KUKA KRL program: MyProgram_231().src

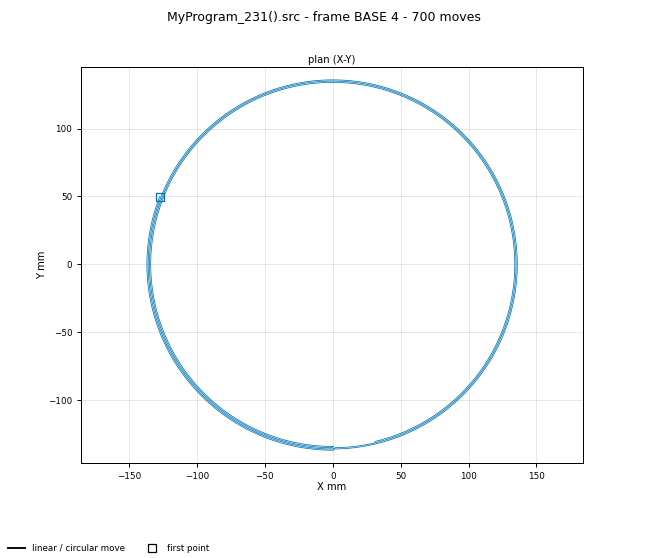
[picture p0: tool path of MyProgram_231().src in frame BASE 4, 700 of 700 moves have a stored position in this frame; points joined in program order, loops and branches not executed]
&ACCESS RVP
&REL 1
&PARAM TEMPLATE = C:\KRC\Roboter\Template\vorgabe
&PARAM EDITMASK = *
DEF MyProgram_231()
; ---- Setting reference (Base) ----
$BASE = BASE_DATA[4]

; --------------------------
; ---- Setting tool (TCP) ----
$TOOL = TOOL_DATA[3]
; --------------------------

$VEL.CP = VEL_APROX_PRINT
Startdeposition()
$VEL.CP = VEL_PRINT
LIN {X -127.3745,Y 49.9123,Z 158,A 155.4211,B 24.9582,C -1.4929,E1 24.8505,E2 291.1488} C_DIS
LIN {X -128.4799,Y 46.9966,Z 158,A 156.8322,B 24.9582,C -1.4941,E1 24.8491,E2 289.7271} C_DIS
LIN {X -130.1138,Y 42.2637,Z 158,A 158.8681,B 24.9587,C -1.4842,E1 24.8473,E2 287.7029} C_DIS
LIN {X -131.1004,Y 39.0966,Z 158,A 160.3394,B 24.9587,C -1.4839,E1 24.8461,E2 286.224} C_DIS
LIN {X -132.2192,Y 35.1211,Z 158,A 161.9803,B 24.9593,C -1.4738,E1 24.8449,E2 284.5976} C_DIS
LIN {X -133.0966,Y 31.6367,Z 158,A 163.554,B 24.9593,C -1.4724,E1 24.8439,E2 283.0182} C_DIS
LIN {X -133.994,Y 27.5885,Z 158,A 165.3357,B 24.9596,C -1.4689,E1 24.8428,E2 281.2342} C_DIS
LIN {X -134.7246,Y 23.7659,Z 158,A 166.9993,B 24.9598,C -1.4652,E1 24.842,E2 279.5695} C_DIS
LIN {X -135.3385,Y 19.9835,Z 158,A 168.5128,B 24.9603,C -1.4553,E1 24.8414,E2 278.0706} C_DIS
LIN {X -135.7642,Y 16.8509,Z 158,A 169.8487,B 24.9605,C -1.4515,E1 24.8409,E2 276.7357} C_DIS
LIN {X -136.156,Y 13.3069,Z 158,A 171.4307,B 24.9605,C -1.4511,E1 24.8404,E2 275.1454} C_DIS
LIN {X -136.4953,Y 9.2216,Z 158,A 173.2066,B 24.9607,C -1.4483,E1 24.8401,E2 273.3653} C_DIS
LIN {X -136.7019,Y 5.2983,Z 158,A 174.7382,B 24.9613,C -1.4371,E1 24.8399,E2 271.8512} C_DIS
LIN {X -136.7995,Y 1.3383,Z 158,A 176.4739,B 24.9613,C -1.4355,E1 24.8398,E2 270.1089} C_DIS
LIN {X -136.7858,Y -2.2665,Z 158,A 177.9865,B 24.9617,C -1.4306,E1 24.8398,E2 268.5987} C_DIS
LIN {X -136.6643,Y -6.2262,Z 158,A 179.6239,B 24.962,C -1.424,E1 24.84,E2 266.9672} C_DIS
LIN {X -136.4748,Y -9.5029,Z 158,A -178.911,B 24.962,C -1.4241,E1 24.8403,E2 265.4932} C_DIS
LIN {X -136.1015,Y -13.8716,Z 158,A -177.0261,B 24.9622,C -1.4205,E1 24.8408,E2 263.6055} C_DIS
LIN {X -135.632,Y -17.8725,Z 158,A -175.4762,B 24.9629,C -1.4081,E1 24.8413,E2 262.076} C_DIS
LIN {X -135.0766,Y -21.687,Z 158,A -173.7107,B 24.9627,C -1.4105,E1 24.8421,E2 260.2943} C_DIS
LIN {X -134.5265,Y -24.8732,Z 158,A -172.3224,B 24.9629,C -1.4078,E1 24.8428,E2 258.904} C_DIS
LIN {X -133.6444,Y -29.2358,Z 158,A -170.5745,B 24.9635,C -1.396,E1 24.8438,E2 257.174} C_DIS
LIN {X -132.6945,Y -33.2823,Z 158,A -168.7848,B 24.9637,C -1.393,E1 24.8449,E2 255.3811} C_DIS
LIN {X -130.9297,Y -39.6606,Z 158,A -166.0195,B 24.9641,C -1.3839,E1 24.8471,E2 252.6213} C_DIS
LIN {X -129.8846,Y -42.9585,Z 158,A -164.5726,B 24.9644,C -1.3794,E1 24.8483,E2 251.1769} C_DIS
LIN {X -128.7046,Y -46.3735,Z 158,A -163.0102,B 24.9644,C -1.3773,E1 24.8498,E2 249.6107} C_DIS
LIN {X -127.0686,Y -50.6869,Z 158,A -161.1504,B 24.965,C -1.3677,E1 24.8516,E2 247.7632} C_DIS
LIN {X -125.8439,Y -53.6576,Z 158,A -159.7893,B 24.9651,C -1.3645,E1 24.8531,E2 246.4022} C_DIS
LIN {X -121.9807,Y -61.9359,Z 158,A -155.9432,B 24.9656,C -1.3543,E1 24.8577,E2 242.5594} C_DIS
LIN {X -119.7997,Y -66.0603,Z 158,A -153.8465,B 24.9656,C -1.3561,E1 24.8605,E2 240.4475} C_DIS
LIN {X -117.4088,Y -70.2217,Z 158,A -151.8184,B 24.9658,C -1.3515,E1 24.8634,E2 238.4198} C_DIS
LIN {X -114.9649,Y -74.1559,Z 158,A -149.8617,B 24.966,C -1.3472,E1 24.8663,E2 236.4634} C_DIS
LIN {X -112.5613,Y -77.756,Z 158,A -148.04,B 24.9662,C -1.3429,E1 24.8691,E2 234.643} C_DIS
LIN {X -109.8954,Y -81.4797,Z 158,A -146.1227,B 24.9665,C -1.338,E1 24.8723,E2 232.7281} C_DIS
LIN {X -107.338,Y -84.8209,Z 158,A -144.3319,B 24.9666,C -1.3351,E1 24.8754,E2 230.9357} C_DIS
LIN {X -104.393,Y -88.4196,Z 158,A -142.0462,B 24.966,C -1.348,E1 24.8795,E2 228.6087} C_DIS
LIN {X -101.6067,Y -91.6087,Z 158,A -140.6091,B 24.9671,C -1.3263,E1 24.8821,E2 227.2167} C_DIS
LIN {X -98.4941,Y -94.9467,Z 158,A -138.4408,B 24.9666,C -1.3354,E1 24.8864,E2 225.0174} C_DIS
LIN {X -95.9147,Y -97.5514,Z 158,A -137.1932,B 24.9675,C -1.3171,E1 24.8888,E2 223.8082} C_DIS
LIN {X -92.7603,Y -100.5557,Z 158,A -135.4258,B 24.9678,C -1.3103,E1 24.8924,E2 222.0497} C_DIS
LIN {X -85.315,Y -106.945,Z 158,A -131.294,B 24.9682,C -1.3032,E1 24.9012,E2 217.9188} C_DIS
LIN {X -82.1496,Y -109.3957,Z 158,A -129.5135,B 24.9681,C -1.3056,E1 24.9051,E2 216.1262} C_DIS
LIN {X -78.4965,Y -112.0463,Z 158,A -127.6003,B 24.9681,C -1.3035,E1 24.9095,E2 214.2114} C_DIS
LIN {X -74.8596,Y -114.5081,Z 158,A -125.7445,B 24.9683,C -1.3014,E1 24.9138,E2 212.3545} C_DIS
LIN {X -71.0332,Y -116.9198,Z 158,A -123.9031,B 24.9686,C -1.2956,E1 24.9182,E2 210.521} C_DIS
LIN {X -67.4593,Y -119.0179,Z 158,A -122.1621,B 24.9686,C -1.2934,E1 24.9224,E2 208.7802} C_DIS
LIN {X -63.8309,Y -121,Z 158,A -120.5227,B 24.969,C -1.2862,E1 24.9264,E2 207.1533} C_DIS
LIN {X -60.8744,Y -122.5145,Z 158,A -119.0759,B 24.969,C -1.2873,E1 24.93,E2 205.6999} C_DIS
LIN {X -51.1886,Y -126.8664,Z 158,A -114.6733,B 24.9693,C -1.2798,E1 24.9413,E2 201.3046} C_DIS
LIN {X -47.6136,Y -128.2516,Z 158,A -112.9917,B 24.9693,C -1.2823,E1 24.9457,E2 199.6137} C_DIS
LIN {X -43.4067,Y -129.7354,Z 158,A -111.2356,B 24.9696,C -1.2746,E1 24.9503,E2 197.8723} C_DIS
LIN {X -40.213,Y -130.7606,Z 158,A -109.8746,B 24.9697,C -1.2712,E1 24.9539,E2 196.517} C_DIS
LIN {X -37.5338,Y -131.5565,Z 158,A -108.4891,B 24.9692,C -1.2819,E1 24.9577,E2 195.1038} C_DIS
LIN {X -33.8507,Y -132.5503,Z 158,A -106.9831,B 24.9695,C -1.276,E1 24.9617,E2 193.6096} C_DIS
LIN {X -30.4717,Y -133.3675,Z 158,A -105.5552,B 24.9696,C -1.2737,E1 24.9656,E2 192.1852} C_DIS
LIN {X -27.3724,Y -134.038,Z 158,A -104.1952,B 24.9696,C -1.2748,E1 24.9693,E2 190.821} C_DIS
LIN {X -23.966,Y -134.6888,Z 158,A -102.7439,B 24.9696,C -1.2742,E1 24.9733,E2 189.3695} C_DIS
LIN {X -19.992,Y -135.3373,Z 158,A -100.9635,B 24.9694,C -1.2788,E1 24.9782,E2 187.5768} C_DIS
LIN {X -11.9765,Y -136.28,Z 158,A -97.5382,B 24.9693,C -1.2808,E1 24.9878,E2 184.1446} C_DIS
LIN {X -7.2873,Y -136.611,Z 158,A -95.6653,B 24.9695,C -1.2756,E1 24.9929,E2 182.2833} C_DIS
LIN {X 0.1481,Y -136.8059,Z 158,A -92.6859,B 24.9699,C -1.2686,E1 25.0012,E2 179.3202} C_DIS
LIN {X 0.1481,Y -136.8059,Z 158,A -92.6859,B 24.9699,C -1.2686,E1 25.0012,E2 179.3202} C_DIS
Enddeposition()
LIN {X 0.9433,Y -135.864,Z 158,A -91.8366,B 24.2391,C -1.1592,E1 24.2683,E2 178.6405} C_DIS
Startdeposition()
$VEL.CP = VEL_PRINT
LIN {X -4.3433,Y -135.807,Z 158,A -94.8507,B 24.241,C -1.1174,E1 24.2596,E2 181.7565} C_DIS
LIN {X -7.4971,Y -135.6699,Z 158,A -96.5948,B 24.2419,C -1.096,E1 24.2546,E2 183.5533} C_DIS
LIN {X -11.0273,Y -135.4276,Z 158,A -97.7763,B 24.2412,C -1.112,E1 24.2514,E2 184.6963} C_DIS
LIN {X -15.1641,Y -135.0278,Z 158,A -99.4494,B 24.241,C -1.1163,E1 24.2467,E2 186.3599} C_DIS
LIN {X -18.8588,Y -134.5605,Z 158,A -101.1029,B 24.2412,C -1.1124,E1 24.2421,E2 188.0243} C_DIS
LIN {X -22.4613,Y -134.0057,Z 158,A -102.5865,B 24.2411,C -1.1156,E1 24.2381,E2 189.5014} C_DIS
LIN {X -25.8541,Y -133.393,Z 158,A -104.0291,B 24.2411,C -1.1167,E1 24.2341,E2 190.9429} C_DIS
LIN {X -29.7466,Y -132.5799,Z 158,A -105.7981,B 24.2411,C -1.1128,E1 24.2292,E2 192.7237} C_DIS
LIN {X -33.6182,Y -131.6505,Z 158,A -107.339,B 24.2408,C -1.1208,E1 24.2251,E2 194.2473} C_DIS
LIN {X -36.7276,Y -130.817,Z 158,A -108.7487,B 24.2409,C -1.119,E1 24.2213,E2 195.6636} C_DIS
LIN {X -39.7605,Y -129.9272,Z 158,A -110.1344,B 24.2409,C -1.1173,E1 24.2176,E2 197.0559} C_DIS
LIN {X -43.4862,Y -128.7294,Z 158,A -111.7492,B 24.2409,C -1.1204,E1 24.2133,E2 198.6661} C_DIS
LIN {X -47.3237,Y -127.3678,Z 158,A -113.58,B 24.241,C -1.1162,E1 24.2085,E2 200.511} C_DIS
LIN {X -51.0417,Y -125.9237,Z 158,A -115.147,B 24.2407,C -1.1237,E1 24.2044,E2 202.0632} C_DIS
LIN {X -56.4466,Y -123.5966,Z 158,A -117.6806,B 24.2407,C -1.1238,E1 24.1979,E2 204.6028} C_DIS
LIN {X -58.9215,Y -122.435,Z 158,A -118.8087,B 24.2406,C -1.1265,E1 24.1951,E2 205.7274} C_DIS
LIN {X -62.0587,Y -120.8754,Z 158,A -120.4233,B 24.2408,C -1.1215,E1 24.191,E2 207.3586} C_DIS
LIN {X -66.2441,Y -118.6353,Z 158,A -122.1842,B 24.2402,C -1.1363,E1 24.1868,E2 209.0885} C_DIS
LIN {X -69.0311,Y -117.0352,Z 158,A -124.0916,B 24.2413,C -1.1108,E1 24.182,E2 211.0643} C_DIS
LIN {X -72.4789,Y -114.9316,Z 158,A -125.2628,B 24.24,C -1.1399,E1 24.1794,E2 212.1682} C_DIS
LIN {X -75.4383,Y -113.0112,Z 158,A -126.9217,B 24.2403,C -1.1337,E1 24.1755,E2 213.8477} C_DIS
LIN {X -79.0416,Y -110.521,Z 158,A -128.8017,B 24.2403,C -1.1352,E1 24.1712,E2 215.7307} C_DIS
LIN {X -82.7672,Y -107.7596,Z 158,A -130.7512,B 24.24,C -1.1391,E1 24.1668,E2 217.6781} C_DIS
LIN {X -86.0862,Y -105.1268,Z 158,A -132.9637,B 24.2408,C -1.1215,E1 24.1619,E2 219.9422} C_DIS
LIN {X -89.3998,Y -102.3233,Z 158,A -134.2995,B 24.2396,C -1.1494,E1 24.1593,E2 221.215} C_DIS
LIN {X -91.7357,Y -100.2353,Z 158,A -135.6918,B 24.2396,C -1.1486,E1 24.1564,E2 222.6151} C_DIS
LIN {X -94.8002,Y -97.3424,Z 158,A -137.6191,B 24.2398,C -1.145,E1 24.1524,E2 224.5595} C_DIS
LIN {X -97.5363,Y -94.5999,Z 158,A -139.1597,B 24.2394,C -1.1531,E1 24.1495,E2 226.087} C_DIS
LIN {X -100.5896,Y -91.3466,Z 158,A -140.8497,B 24.2388,C -1.1668,E1 24.1463,E2 227.7514} C_DIS
LIN {X -103.1897,Y -88.3994,Z 158,A -142.447,B 24.2385,C -1.1736,E1 24.1434,E2 229.3394} C_DIS
LIN {X -105.0465,Y -86.1845,Z 158,A -143.9545,B 24.239,C -1.1623,E1 24.1406,E2 230.8816} C_DIS
LIN {X -107.7192,Y -82.82,Z 158,A -145.7316,B 24.2387,C -1.1685,E1 24.1376,E2 232.6523} C_DIS
LIN {X -110.2344,Y -79.4416,Z 158,A -147.5571,B 24.2387,C -1.1706,E1 24.1346,E2 234.482} C_DIS
LIN {X -112.8321,Y -75.7066,Z 158,A -149.4286,B 24.2383,C -1.1778,E1 24.1316,E2 236.3453} C_DIS
LIN {X -115.1536,Y -72.1268,Z 158,A -151.3159,B 24.2383,C -1.1783,E1 24.1288,E2 238.2412} C_DIS
LIN {X -117.4611,Y -68.3039,Z 158,A -153.1357,B 24.2379,C -1.1865,E1 24.1262,E2 240.0507} C_DIS
LIN {X -119.5108,Y -64.6512,Z 158,A -154.9705,B 24.2379,C -1.1881,E1 24.1237,E2 241.8916} C_DIS
LIN {X -121.3306,Y -61.1645,Z 158,A -157.0591,B 24.2385,C -1.1721,E1 24.121,E2 244.0309} C_DIS
LIN {X -123.2843,Y -57.1221,Z 158,A -158.5479,B 24.2374,C -1.197,E1 24.1193,E2 245.4672} C_DIS
LIN {X -125.3597,Y -52.4109,Z 158,A -160.6334,B 24.2369,C -1.2075,E1 24.117,E2 247.5389} C_DIS
LIN {X -126.641,Y -49.2343,Z 158,A -162.055,B 24.2367,C -1.2129,E1 24.1156,E2 248.9555} C_DIS
LIN {X -127.8904,Y -45.8918,Z 158,A -163.5819,B 24.2365,C -1.2164,E1 24.1141,E2 250.4828} C_DIS
LIN {X -129.0299,Y -42.584,Z 158,A -165.0409,B 24.2363,C -1.2216,E1 24.1128,E2 251.9375} C_DIS
LIN {X -130.1167,Y -39.1413,Z 158,A -166.7844,B 24.2365,C -1.2157,E1 24.1113,E2 253.706} C_DIS
LIN {X -131.5179,Y -34.1405,Z 158,A -168.919,B 24.2361,C -1.2252,E1 24.1098,E2 255.8303} C_DIS
LIN {X -132.4397,Y -30.3603,Z 158,A -171.3415,B 24.2376,C -1.1933,E1 24.1083,E2 258.3455} C_DIS
LIN {X -133.7223,Y -24.0915,Z 158,A -172.9098,B 24.2346,C -1.2556,E1 24.1075,E2 259.7708} C_DIS
LIN {X -134.4968,Y -19.3041,Z 158,A -175.2508,B 24.235,C -1.2479,E1 24.1064,E2 262.1449} C_DIS
LIN {X -134.9819,Y -15.5634,Z 158,A -176.803,B 24.2347,C -1.2549,E1 24.1059,E2 263.6896} C_DIS
LIN {X -135.3593,Y -11.8351,Z 158,A -178.5022,B 24.2347,C -1.2544,E1 24.1055,E2 265.4008} C_DIS
LIN {X -135.6467,Y -7.8912,Z 158,A 179.81,B 24.2345,C -1.2588,E1 24.1052,E2 267.0881} C_DIS
LIN {X -135.8266,Y -3.6367,Z 158,A 178.0552,B 24.2341,C -1.2667,E1 24.105,E2 268.8346} C_DIS
LIN {X -135.8751,Y 0.516,Z 158,A 176.2453,B 24.2339,C -1.2696,E1 24.105,E2 270.6485} C_DIS
LIN {X -135.7956,Y 4.6903,Z 158,A 174.4506,B 24.2337,C -1.2738,E1 24.105,E2 272.4442} C_DIS
LIN {X -135.6064,Y 8.5453,Z 158,A 172.9117,B 24.2333,C -1.2834,E1 24.1053,E2 273.9692} C_DIS
LIN {X -135.2905,Y 12.5973,Z 158,A 171.0922,B 24.2333,C -1.284,E1 24.1058,E2 275.7985} C_DIS
LIN {X -134.9148,Y 16.1259,Z 158,A 169.6758,B 24.2328,C -1.2927,E1 24.1062,E2 277.2023} C_DIS
LIN {X -134.452,Y 19.6178,Z 158,A 168.0516,B 24.2328,C -1.291,E1 24.1068,E2 278.8409} C_DIS
LIN {X -133.7735,Y 23.8054,Z 158,A 166.3023,B 24.2325,C -1.2987,E1 24.1077,E2 280.5819} C_DIS
LIN {X -132.9412,Y 28.0892,Z 158,A 164.2887,B 24.2325,C -1.2965,E1 24.1088,E2 282.6133} C_DIS
LIN {X -132.0076,Y 32.1886,Z 158,A 162.764,B 24.2317,C -1.314,E1 24.1097,E2 284.1042} C_DIS
LIN {X -131.1428,Y 35.5511,Z 158,A 161.1833,B 24.2317,C -1.3132,E1 24.1109,E2 285.6966} C_DIS
LIN {X -130.0069,Y 39.5,Z 158,A 158.8875,B 24.2328,C -1.2921,E1 24.1128,E2 288.0577} C_DIS
LIN {X -128.4489,Y 44.3046,Z 158,A 157.6177,B 24.2304,C -1.3397,E1 24.1138,E2 289.2184} C_DIS
LIN {X -127.1176,Y 47.9918,Z 158,A 155.7295,B 24.2307,C -1.3336,E1 24.1157,E2 291.1325} C_DIS
LIN {X -125.9221,Y 51.0456,Z 158,A 154.3285,B 24.2305,C -1.3371,E1 24.1171,E2 292.533} C_DIS
LIN {X -124.6165,Y 54.1548,Z 158,A 152.8981,B 24.2303,C -1.3411,E1 24.1187,E2 293.9618} C_DIS
LIN {X -123.282,Y 57.1271,Z 158,A 151.4678,B 24.2303,C -1.3426,E1 24.1203,E2 295.3965} C_DIS
LIN {X -121.6635,Y 60.4988,Z 158,A 149.8079,B 24.2302,C -1.3435,E1 24.1224,E2 297.0636} C_DIS
LIN {X -119.5274,Y 64.6204,Z 158,A 147.8581,B 24.2299,C -1.3497,E1 24.1249,E2 299.0089} C_DIS
LIN {X -117.3946,Y 68.4189,Z 158,A 146.0011,B 24.2296,C -1.3541,E1 24.1275,E2 300.865} C_DIS
LIN {X -115.0946,Y 72.2208,Z 158,A 144.079,B 24.2295,C -1.3572,E1 24.1303,E2 302.7896} C_DIS
LIN {X -112.635,Y 75.9991,Z 158,A 142.184,B 24.2292,C -1.363,E1 24.1332,E2 304.6805} C_DIS
LIN {X -109.6094,Y 80.3012,Z 158,A 139.3751,B 24.2303,C -1.341,E1 24.1379,E2 307.5574} C_DIS
LIN {X -106.3504,Y 84.5699,Z 158,A 137.6913,B 24.2285,C -1.3748,E1 24.1407,E2 309.1666} C_DIS
LIN {X -103.4927,Y 88.0439,Z 158,A 135.4483,B 24.2292,C -1.3632,E1 24.1448,E2 311.4486} C_DIS
LIN {X -100.8375,Y 91.0733,Z 158,A 133.9332,B 24.2285,C -1.3763,E1 24.1476,E2 312.9385} C_DIS
LIN {X -97.2173,Y 94.9282,Z 158,A 131.8155,B 24.2279,C -1.3873,E1 24.1516,E2 315.0388} C_DIS
LIN {X -94.0704,Y 98.0474,Z 158,A 129.835,B 24.2279,C -1.3865,E1 24.1556,E2 317.03} C_DIS
LIN {X -89.6733,Y 102.0848,Z 158,A 127.6809,B 24.2266,C -1.4099,E1 24.16,E2 319.1356} C_DIS
LIN {X -87.4419,Y 104.0019,Z 158,A 126.185,B 24.2272,C -1.4004,E1 24.1632,E2 320.6609} C_DIS
LIN {X -84.2261,Y 106.6235,Z 158,A 124.2846,B 24.2274,C -1.3969,E1 24.1674,E2 322.5771} C_DIS
LIN {X -78.8072,Y 110.6886,Z 158,A 121.7162,B 24.2263,C -1.4169,E1 24.1731,E2 325.1059} C_DIS
LIN {X -75.5911,Y 112.9092,Z 158,A 119.8124,B 24.2268,C -1.4078,E1 24.1776,E2 327.0387} C_DIS
LIN {X -69.9156,Y 116.5093,Z 158,A 117.1753,B 24.2259,C -1.4228,E1 24.1837,E2 329.6477} C_DIS
LIN {X -66.69,Y 118.3847,Z 158,A 115.467,B 24.2261,C -1.419,E1 24.1879,E2 331.3705} C_DIS
LIN {X -62.8827,Y 120.4483,Z 158,A 113.7331,B 24.2257,C -1.4267,E1 24.1921,E2 333.0907} C_DIS
LIN {X -59.7011,Y 122.0571,Z 158,A 112.2463,B 24.2255,C -1.4299,E1 24.1959,E2 334.5735} C_DIS
LIN {X -56.8431,Y 123.4133,Z 158,A 110.9005,B 24.2255,C -1.4314,E1 24.1993,E2 335.9192} C_DIS
LIN {X -53.8044,Y 124.768,Z 158,A 109.5225,B 24.2253,C -1.4348,E1 24.2028,E2 337.2924} C_DIS
LIN {X -50.7029,Y 126.0602,Z 158,A 108.063,B 24.2253,C -1.4347,E1 24.2065,E2 338.7556} C_DIS
LIN {X -47.4082,Y 127.3361,Z 158,A 106.555,B 24.2253,C -1.4358,E1 24.2105,E2 340.2641} C_DIS
LIN {X -43.7943,Y 128.6258,Z 158,A 104.7225,B 24.2257,C -1.4272,E1 24.2154,E2 342.1213} C_DIS
LIN {X -38.2828,Y 130.3703,Z 158,A 102.3176,B 24.2254,C -1.4316,E1 24.2218,E2 344.5196} C_DIS
LIN {X -33.519,Y 131.6757,Z 158,A 100.4059,B 24.2249,C -1.4423,E1 24.2269,E2 346.4082} C_DIS
LIN {X -29.9337,Y 132.5371,Z 158,A 98.7925,B 24.2249,C -1.4408,E1 24.2313,E2 348.0275} C_DIS
LIN {X -25.812,Y 133.4011,Z 158,A 97.0468,B 24.2248,C -1.4438,E1 24.2361,E2 349.768} C_DIS
LIN {X -22.3015,Y 134.0324,Z 158,A 95.5753,B 24.2246,C -1.4465,E1 24.2401,E2 351.2342} C_DIS
LIN {X -19.0919,Y 134.5271,Z 158,A 94.1744,B 24.2246,C -1.4459,E1 24.244,E2 352.638} C_DIS
LIN {X -15.0369,Y 135.0415,Z 158,A 92.3855,B 24.2248,C -1.4436,E1 24.2489,E2 354.4338} C_DIS
LIN {X -11.1755,Y 135.4151,Z 158,A 90.7701,B 24.2247,C -1.4454,E1 24.2534,E2 356.0455} C_DIS
LIN {X -6.9273,Y 135.6986,Z 158,A 89.013,B 24.2245,C -1.448,E1 24.2583,E2 357.7968} C_DIS
LIN {X -2.8851,Y 135.8461,Z 158,A 87.2269,B 24.2247,C -1.4444,E1 24.2633,E2 359.5919} C_DIS
LIN {X 0.9988,Y 135.8718,Z 158,A 85.6669,B 24.2245,C -1.4487,E1 24.2676,E2 361.1415} C_DIS
LIN {X 5.2173,Y 135.7751,Z 158,A 83.8781,B 24.2245,C -1.4484,E1 24.2726,E2 362.9307} C_DIS
LIN {X 9.1926,Y 135.5657,Z 158,A 82.106,B 24.2248,C -1.4436,E1 24.2776,E2 364.7137} C_DIS
LIN {X 13.2342,Y 135.2293,Z 158,A 80.5418,B 24.2244,C -1.4509,E1 24.2819,E2 366.2592} C_DIS
LIN {X 16.9507,Y 134.8155,Z 158,A 78.8389,B 24.2248,C -1.4441,E1 24.2867,E2 367.9773} C_DIS
LIN {X 20.7489,Y 134.2815,Z 158,A 77.3159,B 24.2245,C -1.4485,E1 24.2908,E2 369.4882} C_DIS
LIN {X 24.3373,Y 133.6783,Z 158,A 75.8136,B 24.2245,C -1.4495,E1 24.295,E2 370.9863} C_DIS
LIN {X 28.0483,Y 132.95,Z 158,A 74.114,B 24.2248,C -1.4434,E1 24.2997,E2 372.6987} C_DIS
LIN {X 31.9645,Y 132.0617,Z 158,A 72.5449,B 24.2245,C -1.4488,E1 24.3039,E2 374.2522} C_DIS
LIN {X 35.2518,Y 131.2226,Z 158,A 71.0818,B 24.2246,C -1.4462,E1 24.3078,E2 375.7193} C_DIS
LIN {X 38.8483,Y 130.2047,Z 158,A 69.5227,B 24.2246,C -1.4459,E1 24.312,E2 377.2763} C_DIS
LIN {X 41.5644,Y 129.3616,Z 158,A 68.2547,B 24.2249,C -1.4414,E1 24.3154,E2 378.553} C_DIS
LIN {X 46.3316,Y 127.7318,Z 158,A 66.19,B 24.2249,C -1.4426,E1 24.3208,E2 380.6105} C_DIS
LIN {X 49.4364,Y 126.5624,Z 158,A 64.2513,B 24.2265,C -1.4132,E1 24.3261,E2 382.6163} C_DIS
LIN {X 53.681,Y 124.8209,Z 158,A 62.7734,B 24.2253,C -1.4348,E1 24.3297,E2 384.0382} C_DIS
LIN {X 57.3831,Y 123.1636,Z 158,A 61.1802,B 24.225,C -1.4388,E1 24.3337,E2 385.6173} C_DIS
LIN {X 60.1539,Y 121.8336,Z 158,A 59.9125,B 24.225,C -1.4387,E1 24.3369,E2 386.8819} C_DIS
LIN {X 63.4189,Y 120.1667,Z 158,A 58.3725,B 24.2252,C -1.4369,E1 24.3407,E2 388.4217} C_DIS
LIN {X 66.7244,Y 118.3654,Z 158,A 56.4413,B 24.2263,C -1.4166,E1 24.3455,E2 390.3965} C_DIS
LIN {X 69.5862,Y 116.7058,Z 158,A 55.3014,B 24.2257,C -1.4279,E1 24.3482,E2 391.5054} C_DIS
LIN {X 73.2002,Y 114.4736,Z 158,A 53.4864,B 24.2259,C -1.4238,E1 24.3525,E2 393.3244} C_DIS
LIN {X 76.8487,Y 112.0569,Z 158,A 51.6332,B 24.2261,C -1.4202,E1 24.3568,E2 395.1796} C_DIS
LIN {X 80.5046,Y 109.4599,Z 158,A 50.0059,B 24.2255,C -1.4309,E1 24.3604,E2 396.7752} C_DIS
LIN {X 83.0736,Y 107.5234,Z 158,A 47.4593,B 24.229,C -1.3657,E1 24.3664,E2 399.4704} C_DIS
LIN {X 88.6758,Y 102.9517,Z 158,A 45.3805,B 24.2266,C -1.4107,E1 24.3706,E2 401.4315} C_DIS
LIN {X 92.033,Y 99.962,Z 158,A 43.5821,B 24.2266,C -1.412,E1 24.3743,E2 403.2193} C_DIS
LIN {X 95.5132,Y 96.6428,Z 158,A 41.4408,B 24.2271,C -1.4016,E1 24.3786,E2 405.3768} C_DIS
LIN {X 98.6464,Y 93.4421,Z 158,A 39.7077,B 24.2269,C -1.4057,E1 24.3819,E2 407.0921} C_DIS
LIN {X 102.0202,Y 89.7466,Z 158,A 37.5355,B 24.2273,C -1.3975,E1 24.386,E2 409.2742} C_DIS
LIN {X 104.5468,Y 86.7897,Z 158,A 35.8469,B 24.2277,C -1.391,E1 24.389,E2 410.9707} C_DIS
LIN {X 107.3415,Y 83.3083,Z 158,A 34.0218,B 24.2277,C -1.3894,E1 24.3922,E2 412.7907} C_DIS
LIN {X 110.357,Y 79.2704,Z 158,A 31.201,B 24.23,C -1.3467,E1 24.397,E2 415.7009} C_DIS
LIN {X 113.6132,Y 74.5289,Z 158,A 29.4892,B 24.2283,C -1.3786,E1 24.3995,E2 417.3266} C_DIS
LIN {X 115.8811,Y 70.9511,Z 158,A 27.6899,B 24.2286,C -1.3731,E1 24.4022,E2 419.1298} C_DIS
LIN {X 118.1024,Y 67.1886,Z 158,A 25.8524,B 24.2289,C -1.3683,E1 24.4047,E2 420.969} C_DIS
LIN {X 120.1505,Y 63.4499,Z 158,A 24.1116,B 24.2289,C -1.3664,E1 24.407,E2 422.7051} C_DIS
LIN {X 122.9655,Y 57.8112,Z 158,A 21.5099,B 24.2292,C -1.3618,E1 24.4102,E2 425.3036} C_DIS
LIN {X 124.7023,Y 53.9562,Z 158,A 19.7304,B 24.2295,C -1.3568,E1 24.4123,E2 427.0852} C_DIS
LIN {X 125.9943,Y 50.8664,Z 158,A 18.2983,B 24.2298,C -1.3515,E1 24.4138,E2 428.522} C_DIS
LIN {X 127.2874,Y 47.5384,Z 158,A 16.7604,B 24.2301,C -1.3452,E1 24.4153,E2 430.0662} C_DIS
LIN {X 128.642,Y 43.7477,Z 158,A 15.1572,B 24.2301,C -1.3452,E1 24.4168,E2 431.6602} C_DIS
LIN {X 129.612,Y 40.7805,Z 158,A 13.6036,B 24.231,C -1.3282,E1 24.4181,E2 433.2458} C_DIS
LIN {X 130.891,Y 36.463,Z 158,A 11.9512,B 24.2306,C -1.3357,E1 24.4194,E2 434.8702} C_DIS
LIN {X 131.8587,Y 32.7977,Z 158,A 10.2323,B 24.2312,C -1.3241,E1 24.4206,E2 436.607} C_DIS
LIN {X 132.8261,Y 28.6222,Z 158,A 8.6057,B 24.231,C -1.3283,E1 24.4216,E2 438.2136} C_DIS
LIN {X 133.4584,Y 25.5123,Z 158,A 7.2797,B 24.2312,C -1.3247,E1 24.4223,E2 439.5404} C_DIS
LIN {X 134.0223,Y 22.3619,Z 158,A 5.9127,B 24.2314,C -1.3194,E1 24.4229,E2 440.9118} C_DIS
LIN {X 134.5309,Y 19.0656,Z 158,A 4.4948,B 24.2317,C -1.3142,E1 24.4235,E2 442.3337} C_DIS
LIN {X 135.0164,Y 15.2694,Z 158,A 2.78,B 24.2322,C -1.3034,E1 24.4241,E2 444.0641} C_DIS
LIN {X 135.404,Y 11.3066,Z 158,A 1.2125,B 24.2322,C -1.3041,E1 24.4245,E2 445.6204} C_DIS
LIN {X 135.6915,Y 7.0679,Z 158,A -0.6071,B 24.2326,C -1.2967,E1 24.4248,E2 447.4468} C_DIS
LIN {X 135.85,Y 2.6488,Z 158,A -2.4434,B 24.2328,C -1.2921,E1 24.4249,E2 449.2828} C_DIS
LIN {X 135.8706,Y -1.2657,Z 158,A -4.2034,B 24.2334,C -1.2807,E1 24.4249,E2 451.0597} C_DIS
LIN {X 135.7705,Y -5.3351,Z 158,A -5.7294,B 24.2331,C -1.2855,E1 24.4248,E2 452.5647} C_DIS
LIN {X 135.5858,Y -8.8784,Z 158,A -7.3207,B 24.2337,C -1.2753,E1 24.4245,E2 454.1709} C_DIS
LIN {X 135.2428,Y -13.094,Z 158,A -8.9789,B 24.2337,C -1.2763,E1 24.4241,E2 455.8165} C_DIS
LIN {X 134.8417,Y -16.7382,Z 158,A -10.6112,B 24.2341,C -1.2664,E1 24.4236,E2 457.4627} C_DIS
LIN {X 134.2723,Y -20.8082,Z 158,A -12.2869,B 24.2342,C -1.2639,E1 24.4229,E2 459.1343} C_DIS
LIN {X 133.5512,Y -25.0266,Z 158,A -14.1011,B 24.2345,C -1.2575,E1 24.422,E2 460.9531} C_DIS
LIN {X 132.7966,Y -28.7588,Z 158,A -15.602,B 24.2345,C -1.258,E1 24.4212,E2 462.4438} C_DIS
LIN {X 132.0794,Y -31.8909,Z 158,A -16.9691,B 24.2348,C -1.2529,E1 24.4203,E2 463.8149} C_DIS
LIN {X 131.2472,Y -35.1594,Z 158,A -18.3854,B 24.235,C -1.2486,E1 24.4193,E2 465.2332} C_DIS
LIN {X 130.3348,Y -38.4043,Z 158,A -19.8262,B 24.2352,C -1.243,E1 24.4182,E2 466.6792} C_DIS
LIN {X 128.3861,Y -44.4856,Z 158,A -22.1723,B 24.2347,C -1.2535,E1 24.4162,E2 468.9861} C_DIS
LIN {X 126.4013,Y -49.851,Z 158,A -25.3019,B 24.237,C -1.2063,E1 24.413,E2 472.2117} C_DIS
LIN {X 124.9044,Y -53.489,Z 158,A -26.5123,B 24.2361,C -1.2257,E1 24.4118,E2 473.3684} C_DIS
LIN {X 123.2281,Y -57.2436,Z 158,A -28.2493,B 24.2363,C -1.2202,E1 24.4097,E2 475.109} C_DIS
LIN {X 121.6266,Y -60.5737,Z 158,A -29.8033,B 24.2365,C -1.2157,E1 24.4078,E2 476.6654} C_DIS
LIN {X 119.645,Y -64.4015,Z 158,A -31.6763,B 24.2369,C -1.2071,E1 24.4054,E2 478.5489} C_DIS
LIN {X 117.4415,Y -68.3377,Z 158,A -33.6098,B 24.2373,C -1.1998,E1 24.4027,E2 480.4898} C_DIS
LIN {X 114.8464,Y -72.614,Z 158,A -35.6394,B 24.2373,C -1.198,E1 24.3997,E2 482.5131} C_DIS
LIN {X 112.655,Y -75.9696,Z 158,A -37.3341,B 24.2376,C -1.1929,E1 24.3971,E2 484.2114} C_DIS
LIN {X 110.2158,Y -79.4674,Z 158,A -39.1685,B 24.2379,C -1.1858,E1 24.3941,E2 486.0537} C_DIS
LIN {X 107.5431,Y -83.0482,Z 158,A -41.0478,B 24.2382,C -1.1809,E1 24.391,E2 487.9357} C_DIS
LIN {X 104.6303,Y -86.6889,Z 158,A -42.9702,B 24.2382,C -1.178,E1 24.3876,E2 489.8559} C_DIS
LIN {X 101.7935,Y -90.0031,Z 158,A -44.7827,B 24.2384,C -1.1746,E1 24.3843,E2 491.6681} C_DIS
LIN {X 98.2199,Y -93.8899,Z 158,A -47.0302,B 24.2387,C -1.1678,E1 24.38,E2 493.9221} C_DIS
LIN {X 95.6828,Y -96.4743,Z 158,A -48.4971,B 24.2387,C -1.1672,E1 24.3771,E2 495.3838} C_DIS
LIN {X 92.7215,Y -99.3238,Z 158,A -50.1534,B 24.2387,C -1.1672,E1 24.3737,E2 497.0331} C_DIS
LIN {X 89.2983,Y -102.4123,Z 158,A -52.4191,B 24.2398,C -1.1452,E1 24.3689,E2 499.3429} C_DIS
LIN {X 86.7021,Y -104.6194,Z 158,A -53.6265,B 24.2394,C -1.1543,E1 24.3664,E2 500.5234} C_DIS
LIN {X 83.4139,Y -107.2596,Z 158,A -55.391,B 24.2394,C -1.1511,E1 24.3625,E2 502.2888} C_DIS
LIN {X 79.94,Y -109.8732,Z 158,A -57.3575,B 24.24,C -1.14,E1 24.3581,E2 504.2751} C_DIS
LIN {X 76.5471,Y -112.2639,Z 158,A -58.9627,B 24.2398,C -1.1442,E1 24.3544,E2 505.8644} C_DIS
LIN {X 72.8881,Y -114.6733,Z 158,A -60.8391,B 24.24,C -1.139,E1 24.35,E2 507.7472} C_DIS
LIN {X 68.9717,Y -117.0701,Z 158,A -62.6543,B 24.24,C -1.1418,E1 24.3457,E2 509.5496} C_DIS
LIN {X 66.168,Y -118.6778,Z 158,A -64.1037,B 24.2402,C -1.1347,E1 24.3421,E2 511.0119} C_DIS
LIN {X 60.8983,Y -121.4661,Z 158,A -66.4863,B 24.2402,C -1.1374,E1 24.3363,E2 513.381} C_DIS
LIN {X 57.1585,Y -123.2675,Z 158,A -68.0566,B 24.2398,C -1.1442,E1 24.3324,E2 514.9304} C_DIS
LIN {X 55.1738,Y -124.1688,Z 158,A -69.1567,B 24.2403,C -1.1331,E1 24.3295,E2 516.0548} C_DIS
LIN {X 52.0756,Y -125.4997,Z 158,A -70.584,B 24.2403,C -1.1307,E1 24.3258,E2 517.4845} C_DIS
LIN {X 48.4105,Y -126.9607,Z 158,A -72.456,B 24.241,C -1.1172,E1 24.3209,E2 519.3849} C_DIS
LIN {X 44.2917,Y -128.4534,Z 158,A -74.0629,B 24.2405,C -1.1276,E1 24.3167,E2 520.9632} C_DIS
LIN {X 40.836,Y -129.5943,Z 158,A -75.603,B 24.2406,C -1.1254,E1 24.3126,E2 522.5056} C_DIS
LIN {X 37.262,Y -130.6675,Z 158,A -77.4896,B 24.2414,C -1.1071,E1 24.3074,E2 524.4335} C_DIS
LIN {X 34.0289,Y -131.5462,Z 158,A -78.5016,B 24.2406,C -1.1267,E1 24.3048,E2 525.396} C_DIS
LIN {X 29.986,Y -132.5252,Z 158,A -80.3198,B 24.2408,C -1.1217,E1 24.2999,E2 527.224} C_DIS
LIN {X 26.9761,Y -133.1702,Z 158,A -81.6445,B 24.2409,C -1.1191,E1 24.2962,E2 528.5532} C_DIS
LIN {X 23.1292,Y -133.8943,Z 158,A -83.4172,B 24.2412,C -1.1113,E1 24.2913,E2 530.3429} C_DIS
LIN {X 19.3114,Y -134.4958,Z 158,A -84.9171,B 24.241,C -1.117,E1 24.2872,E2 531.8275} C_DIS
LIN {X 15.8599,Y -134.9465,Z 158,A -86.3647,B 24.241,C -1.1171,E1 24.2832,E2 533.2736} C_DIS
LIN {X 11.8233,Y -135.3603,Z 158,A -88.2222,B 24.2414,C -1.1085,E1 24.278,E2 535.1508} C_DIS
LIN {X 8.2925,Y -135.6219,Z 158,A -89.581,B 24.2411,C -1.1149,E1 24.2742,E2 536.4936} C_DIS
LIN {X 4.4841,Y -135.8031,Z 158,A -91.6667,B 24.2422,C -1.0895,E1 24.2683,E2 538.6405} C_DIS
LIN {X 0.9433,Y -135.864,Z 158,A -91.8345,B 24.2392,C -1.1584,E1 24.2683,E2 538.6405} C_DIS
Enddeposition()
LIN {X 0.9433,Y -135.864,Z 158,A -91.8345,B 24.2392,C -1.1584,E1 24.2683,E2 538.6405} C_DIS
Startdeposition()
$VEL.CP = VEL_PRINT
LIN {X 1.7361,Y -134.9358,Z 158,A -91.1259,B 22.6686,C -0.8871,E1 22.6887,E2 538.4231} C_DIS
LIN {X 5.4879,Y -134.8345,Z 158,A -89.4948,B 22.6685,C -0.8894,E1 22.6932,E2 536.7863} C_DIS
LIN {X 10.5137,Y -134.5374,Z 158,A -87.3436,B 22.6685,C -0.891,E1 22.6992,E2 534.6322} C_DIS
LIN {X 14.0292,Y -134.2152,Z 158,A -85.9215,B 22.6685,C -0.888,E1 22.7031,E2 533.2188} C_DIS
LIN {X 17.4825,Y -133.8085,Z 158,A -84.4836,B 22.6685,C -0.8871,E1 22.7071,E2 531.7847} C_DIS
LIN {X 21.2284,Y -133.2669,Z 158,A -82.8212,B 22.6685,C -0.8909,E1 22.7117,E2 530.1141} C_DIS
LIN {X 25.0524,Y -132.6002,Z 158,A -81.247,B 22.6685,C -0.8886,E1 22.716,E2 528.5479} C_DIS
LIN {X 28.41,Y -131.9212,Z 158,A -79.7748,B 22.6685,C -0.8907,E1 22.7201,E2 527.0721} C_DIS
LIN {X 31.8779,Y -131.1266,Z 158,A -78.2556,B 22.6683,C -0.8926,E1 22.7242,E2 525.5505} C_DIS
LIN {X 37.94,Y -129.5024,Z 158,A -74.757,B 22.6666,C -0.9373,E1 22.7339,E2 521.9426} C_DIS
LIN {X 43.9824,Y -127.577,Z 158,A -72.5662,B 22.6675,C -0.9153,E1 22.7395,E2 519.8136} C_DIS
LIN {X 47.4542,Y -126.3265,Z 158,A -71.4662,B 22.6683,C -0.894,E1 22.7423,E2 518.7715} C_DIS
LIN {X 51.5913,Y -124.6948,Z 158,A -69.4682,B 22.668,C -0.9021,E1 22.7475,E2 516.7574} C_DIS
LIN {X 54.8943,Y -123.2758,Z 158,A -68.2123,B 22.6684,C -0.8909,E1 22.7506,E2 515.5341} C_DIS
LIN {X 58.2545,Y -121.7238,Z 158,A -66.2599,B 22.6676,C -0.9124,E1 22.7557,E2 513.5314} C_DIS
LIN {X 62.4355,Y -119.6335,Z 158,A -64.4295,B 22.6678,C -0.9079,E1 22.7602,E2 511.7183} C_DIS
LIN {X 66.1034,Y -117.6483,Z 158,A -62.5549,B 22.6675,C -0.9163,E1 22.7648,E2 509.8283} C_DIS
LIN {X 70.1177,Y -115.3014,Z 158,A -60.5255,B 22.6672,C -0.9227,E1 22.7697,E2 507.7892} C_DIS
LIN {X 74.2418,Y -112.6896,Z 158,A -58.5532,B 22.6672,C -0.9216,E1 22.7743,E2 505.8268} C_DIS
LIN {X 78.0846,Y -110.0623,Z 158,A -56.5498,B 22.667,C -0.927,E1 22.7789,E2 503.8173} C_DIS
LIN {X 81.5243,Y -107.5391,Z 158,A -54.761,B 22.667,C -0.9296,E1 22.7829,E2 502.0287} C_DIS
LIN {X 85.0715,Y -104.7559,Z 158,A -52.9811,B 22.667,C -0.927,E1 22.7867,E2 500.2632} C_DIS
LIN {X 88.6019,Y -101.7866,Z 158,A -50.919,B 22.6667,C -0.9367,E1 22.7912,E2 498.185} C_DIS
LIN {X 91.8184,Y -98.8949,Z 158,A -49.1018,B 22.6665,C -0.94,E1 22.7949,E2 496.3674} C_DIS
LIN {X 94.9926,Y -95.8499,Z 158,A -47.4011,B 22.6667,C -0.936,E1 22.7983,E2 494.685} C_DIS
LIN {X 98.046,Y -92.7243,Z 158,A -45.4309,B 22.6663,C -0.9464,E1 22.8021,E2 492.6973} C_DIS
LIN {X 100.7692,Y -89.758,Z 158,A -43.6834,B 22.666,C -0.9527,E1 22.8054,E2 490.9422} C_DIS
LIN {X 103.6726,Y -86.3884,Z 158,A -41.7776,B 22.6658,C -0.9585,E1 22.8089,E2 489.031} C_DIS
LIN {X 106.5322,Y -82.8355,Z 158,A -39.8711,B 22.6656,C -0.9622,E1 22.8122,E2 487.1252} C_DIS
LIN {X 109.3226,Y -79.1161,Z 158,A -37.926,B 22.6655,C -0.9661,E1 22.8154,E2 485.1805} C_DIS
LIN {X 111.9558,Y -75.3446,Z 158,A -36.2351,B 22.6658,C -0.958,E1 22.818,E2 483.5196} C_DIS
LIN {X 114.4261,Y -71.5369,Z 158,A -34.0463,B 22.6651,C -0.977,E1 22.8214,E2 481.2942} C_DIS
LIN {X 116.8146,Y -67.5659,Z 158,A -32.1702,B 22.6651,C -0.9779,E1 22.824,E2 479.4264} C_DIS
LIN {X 118.8174,Y -63.9783,Z 158,A -30.291,B 22.6645,C -0.99,E1 22.8265,E2 477.5269} C_DIS
LIN {X 120.8884,Y -59.9694,Z 158,A -28.599,B 22.6648,C -0.9842,E1 22.8287,E2 475.86} C_DIS
LIN {X 122.3356,Y -56.9595,Z 158,A -27.1467,B 22.6645,C -0.9902,E1 22.8304,E2 474.4008} C_DIS
LIN {X 125.1785,Y -50.4046,Z 158,A -24.1243,B 22.6641,C -0.9989,E1 22.8337,E2 471.3745} C_DIS
LIN {X 126.5653,Y -46.8168,Z 158,A -22.411,B 22.6638,C -1.0081,E1 22.8354,E2 469.6482} C_DIS
LIN {X 127.8733,Y -43.1156,Z 158,A -20.997,B 22.6641,C -1.0002,E1 22.8367,E2 468.2633} C_DIS
LIN {X 129.2486,Y -38.8023,Z 158,A -18.8782,B 22.6634,C -1.0165,E1 22.8385,E2 466.1161} C_DIS
LIN {X 130.314,Y -35.0521,Z 158,A -17.3145,B 22.6634,C -1.017,E1 22.8396,E2 464.561} C_DIS
LIN {X 131.1636,Y -31.7246,Z 158,A -15.8772,B 22.6632,C -1.0206,E1 22.8406,E2 463.1238} C_DIS
LIN {X 131.9081,Y -28.4708,Z 158,A -14.4551,B 22.663,C -1.0254,E1 22.8414,E2 461.6986} C_DIS
LIN {X 132.7153,Y -24.4429,Z 158,A -12.6768,B 22.6627,C -1.0327,E1 22.8424,E2 459.9128} C_DIS
LIN {X 133.3213,Y -20.8768,Z 158,A -11.2173,B 22.6627,C -1.0337,E1 22.843,E2 458.4602} C_DIS
LIN {X 133.8179,Y -17.4111,Z 158,A -9.7222,B 22.6624,C -1.039,E1 22.8436,E2 456.9614} C_DIS
LIN {X 134.295,Y -13.2423,Z 158,A -7.935,B 22.6622,C -1.0451,E1 22.8441,E2 455.1704} C_DIS
LIN {X 134.6119,Y -9.4941,Z 158,A -6.2706,B 22.6618,C -1.0537,E1 22.8445,E2 453.4947} C_DIS
LIN {X 134.8544,Y -4.9772,Z 158,A -4.5084,B 22.6618,C -1.0518,E1 22.8447,E2 451.7492} C_DIS
LIN {X 134.9426,Y -1.0652,Z 158,A -2.8104,B 22.6616,C -1.059,E1 22.8447,E2 450.0438} C_DIS
LIN {X 134.9172,Y 2.8534,Z 158,A -1.0679,B 22.6611,C -1.0685,E1 22.8447,E2 448.2884} C_DIS
LIN {X 134.7777,Y 6.7354,Z 158,A 0.4772,B 22.6611,C -1.0685,E1 22.8445,E2 446.7537} C_DIS
LIN {X 134.5063,Y 10.8927,Z 158,A 2.2724,B 22.6608,C -1.0755,E1 22.8442,E2 444.9522} C_DIS
LIN {X 134.1485,Y 14.6493,Z 158,A 3.8587,B 22.6606,C -1.0798,E1 22.8437,E2 443.3653} C_DIS
LIN {X 133.5958,Y 19.0401,Z 158,A 5.6561,B 22.6606,C -1.0816,E1 22.843,E2 441.5751} C_DIS
LIN {X 133.0539,Y 22.5191,Z 158,A 7.2289,B 22.6602,C -1.0903,E1 22.8423,E2 439.9901} C_DIS
LIN {X 132.3114,Y 26.5362,Z 158,A 8.8791,B 22.6602,C -1.0914,E1 22.8415,E2 438.3478} C_DIS
LIN {X 131.5935,Y 29.8914,Z 158,A 10.3257,B 22.6599,C -1.0954,E1 22.8406,E2 436.9002} C_DIS
LIN {X 130.7791,Y 33.2737,Z 158,A 11.8213,B 22.6597,C -1.101,E1 22.8396,E2 435.4} C_DIS
LIN {X 129.6441,Y 37.4559,Z 158,A 13.8471,B 22.659,C -1.1162,E1 22.838,E2 433.3479} C_DIS
LIN {X 128.1599,Y 42.255,Z 158,A 15.7548,B 22.6592,C -1.111,E1 22.8364,E2 431.4655} C_DIS
LIN {X 127.2239,Y 45.0001,Z 158,A 17.1191,B 22.6587,C -1.1215,E1 22.8351,E2 430.0827} C_DIS
LIN {X 125.8025,Y 48.8263,Z 158,A 18.7115,B 22.6588,C -1.1195,E1 22.8336,E2 428.5054} C_DIS
LIN {X 124.4635,Y 52.1453,Z 158,A 20.1771,B 22.6588,C -1.1211,E1 22.832,E2 427.0445} C_DIS
LIN {X 123.1173,Y 55.2487,Z 158,A 21.6014,B 22.6586,C -1.1247,E1 22.8304,E2 425.6198} C_DIS
LIN {X 119.8845,Y 61.955,Z 158,A 24.9628,B 22.6577,C -1.1438,E1 22.8262,E2 422.2291} C_DIS
LIN {X 117.6639,Y 66.0757,Z 158,A 26.8115,B 22.6577,C -1.1421,E1 22.8238,E2 420.3955} C_DIS
LIN {X 115.3309,Y 70.0688,Z 158,A 28.7657,B 22.6575,C -1.1469,E1 22.821,E2 418.4401} C_DIS
LIN {X 112.9802,Y 73.7997,Z 158,A 31.0934,B 22.6561,C -1.1751,E1 22.8173,E2 416.0526} C_DIS
LIN {X 110.38,Y 77.6342,Z 158,A 32.569,B 22.6571,C -1.155,E1 22.8151,E2 414.6369} C_DIS
LIN {X 107.9662,Y 80.9583,Z 158,A 34.3492,B 22.6568,C -1.1612,E1 22.8121,E2 412.8503} C_DIS
LIN {X 105.108,Y 84.6352,Z 158,A 36.2997,B 22.6566,C -1.1646,E1 22.8087,E2 410.9012} C_DIS
LIN {X 102.1166,Y 88.2215,Z 158,A 38.0485,B 22.657,C -1.1575,E1 22.8056,E2 409.1798} C_DIS
LIN {X 98.9615,Y 91.7469,Z 158,A 40.2916,B 22.6562,C -1.1738,E1 22.8014,E2 406.9055} C_DIS
LIN {X 95.8225,Y 95.0202,Z 158,A 42.1546,B 22.6562,C -1.1749,E1 22.7977,E2 405.0486} C_DIS
LIN {X 91.96,Y 98.7631,Z 158,A 44.4572,B 22.6559,C -1.1807,E1 22.7931,E2 402.7417} C_DIS
LIN {X 88.5452,Y 101.8361,Z 158,A 46.1298,B 22.6564,C -1.1707,E1 22.7897,E2 401.1024} C_DIS
LIN {X 84.2117,Y 105.4477,Z 158,A 48.7494,B 22.6556,C -1.1864,E1 22.784,E2 398.4531} C_DIS
LIN {X 80.8703,Y 108.032,Z 158,A 50.4745,B 22.6556,C -1.1863,E1 22.7801,E2 396.7355} C_DIS
LIN {X 77.7367,Y 110.3077,Z 158,A 52.2001,B 22.6552,C -1.1932,E1 22.7762,E2 394.9988} C_DIS
LIN {X 73.9323,Y 112.8933,Z 158,A 54.1635,B 22.6551,C -1.1969,E1 22.7716,E2 393.033} C_DIS
LIN {X 70.2768,Y 115.2045,Z 158,A 55.7887,B 22.6554,C -1.1893,E1 22.7678,E2 391.4333} C_DIS
LIN {X 66.5133,Y 117.417,Z 158,A 57.8502,B 22.6548,C -1.2023,E1 22.7628,E2 389.345} C_DIS
LIN {X 63.0552,Y 119.3081,Z 158,A 59.3121,B 22.6552,C -1.1942,E1 22.7592,E2 387.9088} C_DIS
LIN {X 59.8275,Y 120.9585,Z 158,A 60.9253,B 22.6549,C -1.1998,E1 22.7552,E2 386.2859} C_DIS
LIN {X 56.7744,Y 122.4212,Z 158,A 62.3519,B 22.6549,C -1.2011,E1 22.7516,E2 384.8603} C_DIS
LIN {X 51.6246,Y 124.681,Z 158,A 64.7823,B 22.6546,C -1.2058,E1 22.7454,E2 382.4241} C_DIS
LIN {X 47.599,Y 126.2723,Z 158,A 66.494,B 22.6548,C -1.2015,E1 22.7409,E2 380.7278} C_DIS
LIN {X 44.6714,Y 127.3381,Z 158,A 68.1084,B 22.654,C -1.2169,E1 22.7366,E2 379.0771} C_DIS
LIN {X 39.9238,Y 128.9054,Z 158,A 70.1207,B 22.6542,C -1.2133,E1 22.7313,E2 377.0784} C_DIS
LIN {X 36.1818,Y 130.0047,Z 158,A 71.6792,B 22.6544,C -1.2097,E1 22.7271,E2 375.532} C_DIS
LIN {X 32.2714,Y 131.0318,Z 158,A 73.5083,B 22.6541,C -1.2162,E1 22.7221,E2 373.6891} C_DIS
LIN {X 28.3526,Y 131.9336,Z 158,A 75.1235,B 22.6543,C -1.2127,E1 22.7178,E2 372.0855} C_DIS
LIN {X 24.1927,Y 132.7601,Z 158,A 76.9189,B 22.6543,C -1.2132,E1 22.7128,E2 370.2911} C_DIS
LIN {X 20.6757,Y 133.3524,Z 158,A 78.3956,B 22.6543,C -1.2119,E1 22.7088,E2 368.8193} C_DIS
LIN {X 17.4156,Y 133.8173,Z 158,A 79.8366,B 22.6542,C -1.2144,E1 22.7048,E2 367.3734} C_DIS
LIN {X 13.1412,Y 134.3047,Z 158,A 81.579,B 22.6544,C -1.2106,E1 22.7,E2 365.642} C_DIS
LIN {X 9.439,Y 134.6159,Z 158,A 83.331,B 22.6539,C -1.2191,E1 22.695,E2 363.869} C_DIS
LIN {X 5.1396,Y 134.8481,Z 158,A 85.0716,B 22.6541,C -1.2149,E1 22.6902,E2 362.1399} C_DIS
LIN {X 1.1085,Y 134.9419,Z 158,A 86.7892,B 22.6541,C -1.2149,E1 22.6854,E2 360.4225} C_DIS
LIN {X -2.6328,Y 134.9208,Z 158,A 88.4122,B 22.6541,C -1.2162,E1 22.6809,E2 358.7961} C_DIS
LIN {X -6.6879,Y 134.7801,Z 158,A 90.0627,B 22.6543,C -1.2123,E1 22.6763,E2 357.1555} C_DIS
LIN {X -10.5111,Y 134.5376,Z 158,A 91.7594,B 22.6541,C -1.2149,E1 22.6716,E2 355.4512} C_DIS
LIN {X -14.5645,Y 134.1576,Z 158,A 93.458,B 22.6543,C -1.2127,E1 22.6668,E2 353.7574} C_DIS
LIN {X -18.7673,Y 133.6348,Z 158,A 95.2307,B 22.6543,C -1.2104,E1 22.662,E2 351.9891} C_DIS
LIN {X -22.1968,Y 133.1077,Z 158,A 96.6609,B 22.6545,C -1.2074,E1 22.658,E2 350.5653} C_DIS
LIN {X -25.7898,Y 132.4592,Z 158,A 98.3737,B 22.6542,C -1.2138,E1 22.6533,E2 348.8338} C_DIS
LIN {X -29.8311,Y 131.6073,Z 158,A 99.9656,B 22.6547,C -1.2047,E1 22.649,E2 347.2632} C_DIS
LIN {X -33.0534,Y 130.835,Z 158,A 101.4378,B 22.6546,C -1.2065,E1 22.645,E2 345.7843} C_DIS
LIN {X -39.6104,Y 129.0013,Z 158,A 104.3543,B 22.6546,C -1.2046,E1 22.6372,E2 342.8673} C_DIS
LIN {X -43.5903,Y 127.7129,Z 158,A 106.1792,B 22.6546,C -1.2047,E1 22.6323,E2 341.0384} C_DIS
LIN {X -47.028,Y 126.4862,Z 158,A 107.7046,B 22.6548,C -1.2016,E1 22.6283,E2 339.5175} C_DIS
LIN {X -49.8831,Y 125.3887,Z 158,A 109.093,B 22.6547,C -1.204,E1 22.6247,E2 338.1196} C_DIS
LIN {X -53.4935,Y 123.8899,Z 158,A 110.5864,B 22.6552,C -1.194,E1 22.6209,E2 336.6484} C_DIS
LIN {X -56.4744,Y 122.5599,Z 158,A 111.9975,B 22.6552,C -1.1931,E1 22.6173,E2 335.2358} C_DIS
LIN {X -59.3743,Y 121.182,Z 158,A 113.4096,B 22.6552,C -1.1931,E1 22.6138,E2 333.8194} C_DIS
LIN {X -62.3286,Y 119.6896,Z 158,A 114.8251,B 22.6553,C -1.1914,E1 22.6102,E2 332.4044} C_DIS
LIN {X -66.2549,Y 117.5632,Z 158,A 116.7726,B 22.6553,C -1.1905,E1 22.6055,E2 330.4529} C_DIS
LIN {X -71.0341,Y 114.739,Z 158,A 119.2787,B 22.6553,C -1.193,E1 22.5994,E2 327.9316} C_DIS
LIN {X -75.2004,Y 112.0526,Z 158,A 121.2713,B 22.6557,C -1.1838,E1 22.5948,E2 325.9557} C_DIS
LIN {X -78.4662,Y 109.79,Z 158,A 123.3446,B 22.655,C -1.1981,E1 22.59,E2 323.8371} C_DIS
LIN {X -81.8768,Y 107.2706,Z 158,A 124.8016,B 22.656,C -1.1786,E1 22.5869,E2 322.4251} C_DIS
LIN {X -86.2364,Y 103.7985,Z 158,A 127.1241,B 22.6563,C -1.1715,E1 22.5819,E2 320.1114} C_DIS
LIN {X -91.7238,Y 98.983,Z 158,A 130.7762,B 22.6554,C -1.1896,E1 22.5742,E2 316.3959} C_DIS
LIN {X -95.2517,Y 95.5926,Z 158,A 132.3201,B 22.6569,C -1.1603,E1 22.5712,E2 314.9211} C_DIS
LIN {X -97.3039,Y 93.5033,Z 158,A 134.1152,B 22.6558,C -1.1823,E1 22.5676,E2 313.06} C_DIS
LIN {X -100.6203,Y 89.9242,Z 158,A 136.4897,B 22.6554,C -1.1909,E1 22.5632,E2 310.6512} C_DIS
LIN {X -104.8041,Y 85.0119,Z 158,A 138.8855,B 22.6565,C -1.168,E1 22.559,E2 308.3026} C_DIS
LIN {X -107.5875,Y 81.4601,Z 158,A 140.3624,B 22.6577,C -1.143,E1 22.5566,E2 306.8831} C_DIS
LIN {X -110.1696,Y 77.9325,Z 158,A 142.2507,B 22.6579,C -1.1394,E1 22.5535,E2 304.9939} C_DIS
LIN {X -112.7439,Y 74.1592,Z 158,A 144.1819,B 22.6581,C -1.1336,E1 22.5505,E2 303.067} C_DIS
LIN {X -115.1956,Y 70.2913,Z 158,A 146.1609,B 22.6583,C -1.1297,E1 22.5476,E2 301.0872} C_DIS
LIN {X -117.3816,Y 66.5767,Z 158,A 148.0001,B 22.6586,C -1.1248,E1 22.545,E2 299.25} C_DIS
LIN {X -119.416,Y 62.8497,Z 158,A 149.5904,B 22.6592,C -1.11,E1 22.543,E2 297.6888} C_DIS
LIN {X -120.8843,Y 59.9778,Z 158,A 151.0845,B 22.6592,C -1.1115,E1 22.5411,E2 296.1819} C_DIS
LIN {X -122.4216,Y 56.7735,Z 158,A 152.5873,B 22.6594,C -1.1067,E1 22.5393,E2 294.6824} C_DIS
LIN {X -123.8112,Y 53.6755,Z 158,A 154.0265,B 22.6596,C -1.1023,E1 22.5377,E2 293.2461} C_DIS
LIN {X -125.0735,Y 50.6651,Z 158,A 155.4775,B 22.6596,C -1.1009,E1 22.5361,E2 291.7896} C_DIS
LIN {X -126.1642,Y 47.8875,Z 158,A 156.81,B 22.6597,C -1.0999,E1 22.5348,E2 290.4514} C_DIS
LIN {X -127.6172,Y 43.8665,Z 158,A 159.1789,B 22.6588,C -1.1191,E1 22.5326,E2 288.0173} C_DIS
LIN {X -129.1414,Y 39.1525,Z 158,A 160.4458,B 22.6608,C -1.0751,E1 22.5316,E2 286.8573} C_DIS
LIN {X -129.9551,Y 36.3591,Z 158,A 162.1596,B 22.6601,C -1.0925,E1 22.5303,E2 285.0869} C_DIS
LIN {X -131.1284,Y 31.8706,Z 158,A 164.3873,B 22.6598,C -1.0977,E1 22.5288,E2 282.8309} C_DIS
LIN {X -132.0864,Y 27.6419,Z 158,A 165.8724,B 22.6608,C -1.0759,E1 22.5279,E2 281.3931} C_DIS
LIN {X -132.7563,Y 24.2139,Z 158,A 167.2608,B 22.6612,C -1.0669,E1 22.5272,E2 280.0189} C_DIS
LIN {X -133.3505,Y 20.6883,Z 158,A 168.7865,B 22.6614,C -1.0624,E1 22.5265,E2 278.495} C_DIS
LIN {X -133.8381,Y 17.2573,Z 158,A 170.3101,B 22.6615,C -1.06,E1 22.526,E2 276.9675} C_DIS
LIN {X -134.2718,Y 13.4834,Z 158,A 171.9504,B 22.6617,C -1.056,E1 22.5255,E2 275.3268} C_DIS
LIN {X -134.5869,Y 9.8361,Z 158,A 173.4683,B 22.662,C -1.0493,E1 22.5251,E2 273.816} C_DIS
LIN {X -134.8132,Y 6.0299,Z 158,A 175.2223,B 22.662,C -1.0501,E1 22.5249,E2 272.0483} C_DIS
LIN {X -134.9299,Y 2.0899,Z 158,A 176.7644,B 22.6624,C -1.0388,E1 22.5248,E2 270.5251} C_DIS
LIN {X -134.9346,Y -1.8042,Z 158,A 178.5071,B 22.6625,C -1.0375,E1 22.5248,E2 268.7743} C_DIS
LIN {X -134.8298,Y -5.6078,Z 158,A -179.7977,B 22.6625,C -1.0358,E1 22.525,E2 267.072} C_DIS
LIN {X -134.5894,Y -9.8017,Z 158,A -178.1819,B 22.6631,C -1.0226,E1 22.5253,E2 265.4799} C_DIS
LIN {X -134.3295,Y -12.8825,Z 158,A -176.8011,B 22.6631,C -1.0214,E1 22.5256,E2 264.0928} C_DIS
LIN {X -133.9495,Y -16.3724,Z 158,A -175.1895,B 22.6631,C -1.0221,E1 22.5261,E2 262.4688} C_DIS
LIN {X -133.3825,Y -20.4817,Z 158,A -173.527,B 22.6636,C -1.0121,E1 22.5268,E2 260.8213} C_DIS
LIN {X -132.9181,Y -23.3097,Z 158,A -172.0719,B 22.6633,C -1.0189,E1 22.5275,E2 259.3387} C_DIS
LIN {X -130.7202,Y -33.5058,Z 158,A -167.508,B 22.6636,C -1.0112,E1 22.5304,E2 254.7651} C_DIS
LIN {X -129.7939,Y -36.9354,Z 158,A -166.2029,B 22.6642,C -0.9974,E1 22.5313,E2 253.4876} C_DIS
LIN {X -128.6203,Y -40.8309,Z 158,A -164.5753,B 22.6646,C -0.9877,E1 22.5327,E2 251.875} C_DIS
LIN {X -127.5287,Y -44.1216,Z 158,A -163.1421,B 22.6649,C -0.9815,E1 22.5339,E2 250.4486} C_DIS
LIN {X -126.482,Y -47.0393,Z 158,A -161.7044,B 22.6648,C -0.9831,E1 22.5353,E2 248.9979} C_DIS
LIN {X -125.1803,Y -50.4002,Z 158,A -160.2747,B 22.6652,C -0.9741,E1 22.5368,E2 247.5828} C_DIS
LIN {X -123.9776,Y -53.2906,Z 158,A -159.0896,B 22.6656,C -0.9638,E1 22.5381,E2 246.4172} C_DIS
LIN {X -121.9097,Y -57.8654,Z 158,A -156.6687,B 22.6653,C -0.9707,E1 22.5409,E2 243.9635} C_DIS
LIN {X -120.5627,Y -60.6245,Z 158,A -155.2948,B 22.6653,C -0.9702,E1 22.5426,E2 242.5827} C_DIS
LIN {X -118.6191,Y -64.3459,Z 158,A -153.523,B 22.6655,C -0.9648,E1 22.545,E2 240.8145} C_DIS
LIN {X -116.3943,Y -68.2872,Z 158,A -151.6203,B 22.6658,C -0.9587,E1 22.5476,E2 238.9165} C_DIS
LIN {X -113.9677,Y -72.265,Z 158,A -149.6239,B 22.666,C -0.9543,E1 22.5506,E2 236.9203} C_DIS
LIN {X -111.4947,Y -76.0256,Z 158,A -147.6747,B 22.666,C -0.9511,E1 22.5536,E2 234.9685} C_DIS
LIN {X -108.9344,Y -79.6503,Z 158,A -145.7848,B 22.6663,C -0.9467,E1 22.5567,E2 233.08} C_DIS
LIN {X -106.2501,Y -83.197,Z 158,A -143.895,B 22.6664,C -0.9421,E1 22.5599,E2 231.192} C_DIS
LIN {X -103.4018,Y -86.7113,Z 158,A -141.9185,B 22.6665,C -0.9402,E1 22.5634,E2 229.2104} C_DIS
LIN {X -100.2317,Y -90.358,Z 158,A -140.1315,B 22.6672,C -0.9233,E1 22.5666,E2 227.4584} C_DIS
LIN {X -97.9323,Y -92.8448,Z 158,A -138.5658,B 22.6671,C -0.926,E1 22.5697,E2 225.8782} C_DIS
LIN {X -95.1869,Y -95.6569,Z 158,A -136.806,B 22.6671,C -0.9266,E1 22.5731,E2 224.1084} C_DIS
LIN {X -91.9799,Y -98.7445,Z 158,A -134.9041,B 22.6671,C -0.9232,E1 22.577,E2 222.2065} C_DIS
LIN {X -87.4827,Y -102.7501,Z 158,A -132.3437,B 22.6674,C -0.9183,E1 22.5824,E2 219.6477} C_DIS
LIN {X -84.0847,Y -105.5488,Z 158,A -130.4765,B 22.6675,C -0.9147,E1 22.5864,E2 217.782} C_DIS
LIN {X -80.6941,Y -108.1631,Z 158,A -128.6226,B 22.6675,C -0.9131,E1 22.5906,E2 215.9248} C_DIS
LIN {X -76.9249,Y -110.8755,Z 158,A -126.6547,B 22.6677,C -0.9096,E1 22.595,E2 213.9584} C_DIS
LIN {X -73.2088,Y -113.3639,Z 158,A -124.9157,B 22.6681,C -0.8991,E1 22.599,E2 212.2404} C_DIS
LIN {X -66.8374,Y -117.2329,Z 158,A -121.4772,B 22.6678,C -0.9072,E1 22.6074,E2 208.7692} C_DIS
LIN {X -62.7077,Y -119.4905,Z 158,A -119.6801,B 22.6683,C -0.8951,E1 22.6117,E2 206.9981} C_DIS
LIN {X -60.0208,Y -120.8631,Z 158,A -118.3765,B 22.6683,C -0.8945,E1 22.615,E2 205.6921} C_DIS
LIN {X -57.4037,Y -122.1302,Z 158,A -116.8406,B 22.6678,C -0.9072,E1 22.619,E2 204.1187} C_DIS
LIN {X -52.7629,Y -124.2054,Z 158,A -114.8108,B 22.6681,C -0.8988,E1 22.6241,E2 202.1056} C_DIS
LIN {X -49.2283,Y -125.6462,Z 158,A -113.3546,B 22.6685,C -0.8894,E1 22.6278,E2 200.6703} C_DIS
LIN {X -44.8398,Y -127.2797,Z 158,A -111.2829,B 22.6684,C -0.8915,E1 22.6333,E2 198.5884} C_DIS
LIN {X -41.0609,Y -128.5469,Z 158,A -109.653,B 22.6685,C -0.8872,E1 22.6376,E2 196.9663} C_DIS
LIN {X -37.7798,Y -129.5492,Z 158,A -108.1955,B 22.6685,C -0.8862,E1 22.6415,E2 195.5087} C_DIS
LIN {X -34.5827,Y -130.4392,Z 158,A -106.7357,B 22.6685,C -0.8877,E1 22.6455,E2 194.0425} C_DIS
LIN {X -30.2792,Y -131.5049,Z 158,A -104.8827,B 22.6686,C -0.8853,E1 22.6505,E2 192.1931} C_DIS
LIN {X -27.0133,Y -132.2143,Z 158,A -103.4751,B 22.6686,C -0.8841,E1 22.6543,E2 190.7867} C_DIS
LIN {X -23.7357,Y -132.8419,Z 158,A -102.0702,B 22.6687,C -0.883,E1 22.6582,E2 189.3831} C_DIS
LIN {X -20.2796,Y -133.4138,Z 158,A -100.4621,B 22.6685,C -0.8883,E1 22.6627,E2 187.7593} C_DIS
LIN {X -16.085,Y -133.9838,Z 158,A -98.9803,B 22.6691,C -0.8728,E1 22.6666,E2 186.3169} C_DIS
LIN {X -12.4381,Y -134.3722,Z 158,A -97.2255,B 22.6687,C -0.8821,E1 22.6716,E2 184.5367} C_DIS
LIN {X -8.5427,Y -134.6754,Z 158,A -95.485,B 22.6686,C -0.886,E1 22.6765,E2 182.7852} C_DIS
LIN {X -4.1696,Y -134.8822,Z 158,A -93.8608,B 22.669,C -0.8748,E1 22.6809,E2 181.1898} C_DIS
LIN {X -0.7654,Y -134.9438,Z 158,A -92.1219,B 22.6685,C -0.8893,E1 22.6859,E2 179.4132} C_DIS
LIN {X -0.7654,Y -134.9438,Z 158,A -92.1219,B 22.6685,C -0.8893,E1 22.6859,E2 179.4132} C_DIS
Enddeposition()
LIN {X 0.9335,Y -134.0118,Z 158,A -91.4763,B 21.5063,C -0.6964,E1 21.5187,E2 179.1521} C_DIS
Startdeposition()
$VEL.CP = VEL_PRINT
LIN {X -1.4841,Y -134.0105,Z 158,A -92.9578,B 21.507,C -0.6758,E1 21.5144,E2 180.6898} C_DIS
LIN {X -5.2064,Y -133.9154,Z 158,A -94.4474,B 21.5068,C -0.6803,E1 21.5103,E2 182.1674} C_DIS
LIN {X -8.9978,Y -133.7163,Z 158,A -96.0345,B 21.5068,C -0.6818,E1 21.5058,E2 183.7507} C_DIS
LIN {X -11.7404,Y -133.5021,Z 158,A -97.2325,B 21.5068,C -0.681,E1 21.5025,E2 184.9519} C_DIS
LIN {X -16.1,Y -133.0461,Z 158,A -99.1025,B 21.5068,C -0.6814,E1 21.4973,E2 186.822} C_DIS
LIN {X -19.4254,Y -132.602,Z 158,A -100.4997,B 21.5068,C -0.6834,E1 21.4935,E2 188.2149} C_DIS
LIN {X -22.5248,Y -132.1108,Z 158,A -101.8742,B 21.5068,C -0.6824,E1 21.4897,E2 189.5939} C_DIS
LIN {X -25.6351,Y -131.5426,Z 158,A -103.2178,B 21.5068,C -0.6833,E1 21.486,E2 190.9367} C_DIS
LIN {X -28.7033,Y -130.9072,Z 158,A -104.5991,B 21.5068,C -0.682,E1 21.4822,E2 192.3233} C_DIS
LIN {X -31.8772,Y -130.1708,Z 158,A -105.9898,B 21.5068,C -0.6829,E1 21.4784,E2 193.7138} C_DIS
LIN {X -35.0036,Y -129.3652,Z 158,A -107.342,B 21.5067,C -0.685,E1 21.4748,E2 195.0627} C_DIS
LIN {X -38.0492,Y -128.5021,Z 158,A -108.7426,B 21.5067,C -0.6838,E1 21.471,E2 196.4691} C_DIS
LIN {X -41.5615,Y -127.4114,Z 158,A -110.2886,B 21.5067,C -0.6862,E1 21.4669,E2 198.012} C_DIS
LIN {X -44.6772,Y -126.3525,Z 158,A -111.7001,B 21.5067,C -0.6872,E1 21.4632,E2 199.4239} C_DIS
LIN {X -47.6323,Y -125.2675,Z 158,A -113.0296,B 21.5066,C -0.6892,E1 21.4597,E2 200.7513} C_DIS
LIN {X -50.5098,Y -124.1341,Z 158,A -114.407,B 21.5066,C -0.6881,E1 21.4561,E2 202.1352} C_DIS
LIN {X -53.9533,Y -122.6787,Z 158,A -115.9819,B 21.5066,C -0.6908,E1 21.4521,E2 203.7071} C_DIS
LIN {X -56.7089,Y -121.4276,Z 158,A -117.2806,B 21.5065,C -0.6921,E1 21.4488,E2 205.0059} C_DIS
LIN {X -59.7208,Y -119.9748,Z 158,A -118.8477,B 21.5066,C -0.6879,E1 21.4448,E2 206.5895} C_DIS
LIN {X -63.8031,Y -117.8566,Z 158,A -120.8268,B 21.5066,C -0.6899,E1 21.4399,E2 208.5696} C_DIS
LIN {X -67.659,Y -115.6856,Z 158,A -122.6888,B 21.5064,C -0.6939,E1 21.4354,E2 210.4273} C_DIS
LIN {X -71.0264,Y -113.6492,Z 158,A -124.28,B 21.5062,C -0.7004,E1 21.4317,E2 212.0065} C_DIS
LIN {X -74.2861,Y -111.5456,Z 158,A -126.0433,B 21.5062,C -0.6985,E1 21.4275,E2 213.7819} C_DIS
LIN {X -77.9292,Y -109.0315,Z 158,A -127.918,B 21.5062,C -0.7024,E1 21.4232,E2 215.6533} C_DIS
LIN {X -81.5362,Y -106.3611,Z 158,A -129.8131,B 21.506,C -0.7068,E1 21.419,E2 217.5445} C_DIS
LIN {X -84.4717,Y -104.0459,Z 158,A -131.462,B 21.506,C -0.7076,E1 21.4154,E2 219.1986} C_DIS
LIN {X -87.7876,Y -101.2638,Z 158,A -133.3702,B 21.506,C -0.7086,E1 21.4113,E2 221.1124} C_DIS
LIN {X -90.9952,Y -98.3914,Z 158,A -135.1384,B 21.5057,C -0.7154,E1 21.4077,E2 222.8705} C_DIS
LIN {X -94.0276,Y -95.4971,Z 158,A -136.9579,B 21.5057,C -0.718,E1 21.4041,E2 224.6919} C_DIS
LIN {X -97.0681,Y -92.405,Z 158,A -138.8389,B 21.5056,C -0.7209,E1 21.4004,E2 226.5747} C_DIS
LIN {X -100.0057,Y -89.2174,Z 158,A -140.672,B 21.5054,C -0.7259,E1 21.397,E2 228.4037} C_DIS
LIN {X -102.7993,Y -85.9836,Z 158,A -142.5355,B 21.5054,C -0.7285,E1 21.3936,E2 230.2699} C_DIS
LIN {X -105.5555,Y -82.5769,Z 158,A -144.3605,B 21.5051,C -0.735,E1 21.3904,E2 232.0873} C_DIS
LIN {X -107.8513,Y -79.5549,Z 158,A -146.0711,B 21.5051,C -0.7353,E1 21.3876,E2 233.8069} C_DIS
LIN {X -110.3519,Y -76.0484,Z 158,A -147.9225,B 21.505,C -0.7395,E1 21.3846,E2 235.6576} C_DIS
LIN {X -112.5328,Y -72.7823,Z 158,A -149.5789,B 21.5048,C -0.7447,E1 21.3821,E2 237.3094} C_DIS
LIN {X -114.882,Y -69.0152,Z 158,A -151.4844,B 21.5046,C -0.7494,E1 21.3793,E2 239.2136} C_DIS
LIN {X -117.0377,Y -65.2931,Z 158,A -153.2701,B 21.5044,C -0.7565,E1 21.3768,E2 240.9907} C_DIS
LIN {X -118.8264,Y -61.9735,Z 158,A -154.9052,B 21.5043,C -0.76,E1 21.3747,E2 242.6266} C_DIS
LIN {X -120.4136,Y -58.8313,Z 158,A -156.3929,B 21.5041,C -0.7649,E1 21.3728,E2 244.1103} C_DIS
LIN {X -121.9937,Y -55.4848,Z 158,A -157.9973,B 21.5041,C -0.7684,E1 21.3709,E2 245.7154} C_DIS
LIN {X -123.1244,Y -52.9224,Z 158,A -159.2174,B 21.5039,C -0.7709,E1 21.3696,E2 246.9367} C_DIS
LIN {X -124.3978,Y -49.8557,Z 158,A -160.6564,B 21.5039,C -0.7742,E1 21.3681,E2 248.3761} C_DIS
LIN {X -125.6771,Y -46.5388,Z 158,A -162.1345,B 21.5036,C -0.7804,E1 21.3666,E2 249.8471} C_DIS
LIN {X -126.7121,Y -43.6399,Z 158,A -163.4705,B 21.5035,C -0.7834,E1 21.3654,E2 251.1837} C_DIS
LIN {X -127.7425,Y -40.5249,Z 158,A -164.919,B 21.5035,C -0.7857,E1 21.3641,E2 252.6358} C_DIS
LIN {X -128.7549,Y -37.1857,Z 158,A -166.394,B 21.5032,C -0.7909,E1 21.3629,E2 254.1067} C_DIS
LIN {X -129.5944,Y -34.1439,Z 158,A -167.7594,B 21.5032,C -0.7943,E1 21.362,E2 255.4721} C_DIS
LIN {X -130.4729,Y -30.624,Z 158,A -169.3118,B 21.5029,C -0.7989,E1 21.3609,E2 257.0225} C_DIS
LIN {X -131.1665,Y -27.5019,Z 158,A -170.6876,B 21.5029,C -0.8028,E1 21.3601,E2 258.3972} C_DIS
LIN {X -131.7813,Y -24.3865,Z 158,A -172.0532,B 21.5027,C -0.8067,E1 21.3594,E2 259.7617} C_DIS
LIN {X -132.4925,Y -20.156,Z 158,A -173.9335,B 21.5025,C -0.8105,E1 21.3586,E2 261.6447} C_DIS
LIN {X -132.9812,Y -16.6437,Z 158,A -175.4233,B 21.5023,C -0.8163,E1 21.358,E2 263.1291} C_DIS
LIN {X -133.2923,Y -13.9196,Z 158,A -176.627,B 21.5023,C -0.8188,E1 21.3576,E2 264.3347} C_DIS
LIN {X -133.6432,Y -9.9998,Z 158,A -178.35,B 21.5021,C -0.8224,E1 21.3572,E2 266.0598} C_DIS
LIN {X -133.8574,Y -6.5326,Z 158,A -179.7749,B 21.5018,C -0.8296,E1 21.357,E2 267.4751} C_DIS
LIN {X -133.9775,Y -3.271,Z 158,A 178.8082,B 21.5018,C -0.8332,E1 21.357,E2 268.8923} C_DIS
LIN {X -134.0195,Y 0,Z 158,A 177.3846,B 21.5016,C -0.8366,E1 21.3569,E2 270.3168} C_DIS
LIN {X -133.9732,Y 3.4249,Z 158,A 175.8592,B 21.5016,C -0.8388,E1 21.3569,E2 271.847} C_DIS
LIN {X -133.8407,Y 6.866,Z 158,A 174.4082,B 21.5013,C -0.8444,E1 21.3571,E2 273.293} C_DIS
LIN {X -133.6273,Y 10.2166,Z 158,A 172.9843,B 21.5011,C -0.8494,E1 21.3574,E2 274.7131} C_DIS
LIN {X -133.3298,Y 13.5716,Z 158,A 171.5304,B 21.501,C -0.8534,E1 21.3578,E2 276.1664} C_DIS
LIN {X -132.9812,Y 16.6437,Z 158,A 170.1963,B 21.5008,C -0.8571,E1 21.3582,E2 277.4998} C_DIS
LIN {X -132.3184,Y 21.2802,Z 158,A 168.1745,B 21.5006,C -0.8627,E1 21.3591,E2 279.5205} C_DIS
LIN {X -131.8364,Y 24.0787,Z 158,A 166.9485,B 21.5005,C -0.8661,E1 21.3597,E2 280.7458} C_DIS
LIN {X -131.2293,Y 27.1934,Z 158,A 165.5943,B 21.5003,C -0.8705,E1 21.3604,E2 282.0974} C_DIS
LIN {X -130.4729,Y 30.624,Z 158,A 164.064,B 21.5002,C -0.874,E1 21.3613,E2 283.6287} C_DIS
LIN {X -129.8176,Y 33.2845,Z 158,A 162.8644,B 21.5001,C -0.8766,E1 21.3622,E2 284.8295} C_DIS
LIN {X -128.8454,Y 36.8763,Z 158,A 161.2762,B 21.4999,C -0.8816,E1 21.3633,E2 286.4147} C_DIS
LIN {X -127.9099,Y 40.0009,Z 158,A 159.8692,B 21.4997,C -0.8854,E1 21.3645,E2 287.8209} C_DIS
LIN {X -126.8923,Y 43.1203,Z 158,A 158.4539,B 21.4996,C -0.8892,E1 21.3657,E2 289.2353} C_DIS
LIN {X -125.903,Y 45.9239,Z 158,A 157.1506,B 21.4995,C -0.8918,E1 21.367,E2 290.5402} C_DIS
LIN {X -124.609,Y 49.3316,Z 158,A 155.5999,B 21.4993,C -0.8969,E1 21.3685,E2 292.0875} C_DIS
LIN {X -123.3429,Y 52.417,Z 158,A 154.1619,B 21.4991,C -0.9007,E1 21.3701,E2 293.5245} C_DIS
LIN {X -122.2177,Y 54.9839,Z 158,A 152.9292,B 21.4991,C -0.9029,E1 21.3715,E2 294.7592} C_DIS
LIN {X -120.7053,Y 58.2305,Z 158,A 151.3883,B 21.4989,C -0.907,E1 21.3733,E2 296.2987} C_DIS
LIN {X -118.8906,Y 61.8512,Z 158,A 149.6054,B 21.4987,C -0.9099,E1 21.3756,E2 298.0848} C_DIS
LIN {X -116.7428,Y 65.8177,Z 158,A 147.6874,B 21.4985,C -0.9159,E1 21.3782,E2 299.9984} C_DIS
LIN {X -114.6639,Y 69.376,Z 158,A 145.9081,B 21.4983,C -0.9201,E1 21.3807,E2 301.7768} C_DIS
LIN {X -112.7317,Y 72.4739,Z 158,A 144.3071,B 21.4983,C -0.9228,E1 21.3831,E2 303.3801} C_DIS
LIN {X -110.3519,Y 76.0484,Z 158,A 142.5233,B 21.4979,C -0.93,E1 21.3859,E2 305.1547} C_DIS
LIN {X -108.361,Y 78.8593,Z 158,A 140.9746,B 21.4979,C -0.9308,E1 21.3884,E2 306.7101} C_DIS
LIN {X -105.7659,Y 82.3072,Z 158,A 139.1168,B 21.4977,C -0.9352,E1 21.3916,E2 308.5665} C_DIS
LIN {X -103.0556,Y 85.6763,Z 158,A 137.2557,B 21.4975,C -0.9394,E1 21.3948,E2 310.4261} C_DIS
LIN {X -100.2338,Y 88.9611,Z 158,A 135.4584,B 21.4972,C -0.9463,E1 21.3981,E2 312.2141} C_DIS
LIN {X -97.8988,Y 91.5245,Z 158,A 133.901,B 21.4972,C -0.9468,E1 21.4011,E2 313.7782} C_DIS
LIN {X -94.8866,Y 94.6437,Z 158,A 132.0809,B 21.497,C -0.9527,E1 21.4046,E2 315.5914} C_DIS
LIN {X -92.1765,Y 97.2852,Z 158,A 130.3677,B 21.497,C -0.9525,E1 21.4081,E2 317.3136} C_DIS
LIN {X -89.2174,Y 100.0057,Z 158,A 128.747,B 21.4967,C -0.9605,E1 21.4114,E2 318.9202} C_DIS
LIN {X -86.4002,Y 102.4498,Z 158,A 127.0251,B 21.4967,C -0.9586,E1 21.4151,E2 320.655} C_DIS
LIN {X -83.122,Y 105.1273,Z 158,A 125.281,B 21.4964,C -0.9652,E1 21.4189,E2 322.3887} C_DIS
LIN {X -79.8295,Y 107.6483,Z 158,A 123.5513,B 21.4962,C -0.9707,E1 21.4227,E2 324.1108} C_DIS
LIN {X -76.8951,Y 109.7641,Z 158,A 121.8627,B 21.4963,C -0.9678,E1 21.4266,E2 325.8143} C_DIS
LIN {X -73.3363,Y 112.1731,Z 158,A 120.1463,B 21.496,C -0.9764,E1 21.4305,E2 327.5139} C_DIS
LIN {X -70.4435,Y 114.012,Z 158,A 118.6754,B 21.4959,C -0.9788,E1 21.434,E2 328.9835} C_DIS
LIN {X -67.0192,Y 116.0572,Z 158,A 116.9254,B 21.4959,C -0.9799,E1 21.4382,E2 330.7368} C_DIS
LIN {X -63.8031,Y 117.8566,Z 158,A 115.2454,B 21.4959,C -0.9781,E1 21.4424,E2 332.4273} C_DIS
LIN {X -60.5076,Y 119.5794,Z 158,A 113.7867,B 21.4955,C -0.9863,E1 21.4459,E2 333.8684} C_DIS
LIN {X -57.5187,Y 121.0454,Z 158,A 112.361,B 21.4955,C -0.9884,E1 21.4495,E2 335.2927} C_DIS
LIN {X -54.4537,Y 122.4548,Z 158,A 110.8914,B 21.4955,C -0.9893,E1 21.4533,E2 336.7639} C_DIS
LIN {X -51.1813,Y 123.859,Z 158,A 109.3893,B 21.4953,C -0.9923,E1 21.4571,E2 338.262} C_DIS
LIN {X -48.0897,Y 125.0918,Z 158,A 107.9634,B 21.4952,C -0.994,E1 21.4608,E2 339.6867} C_DIS
LIN {X -44.6772,Y 126.3525,Z 158,A 106.4051,B 21.4952,C -0.9958,E1 21.4649,E2 341.2439} C_DIS
LIN {X -41.87,Y 127.3086,Z 158,A 105.1354,B 21.4951,C -0.9972,E1 21.4683,E2 342.5125} C_DIS
LIN {X -38.7482,Y 128.2933,Z 158,A 103.734,B 21.495,C -0.9987,E1 21.472,E2 343.9128} C_DIS
LIN {X -35.6226,Y 129.1961,Z 158,A 102.3671,B 21.4949,C -1.0012,E1 21.4757,E2 345.2755} C_DIS
LIN {X -32.6806,Y 129.9709,Z 158,A 100.993,B 21.4949,C -0.9992,E1 21.4794,E2 346.6572} C_DIS
LIN {X -29.3714,Y 130.759,Z 158,A 99.5647,B 21.4949,C -1.0016,E1 21.4833,E2 348.0813} C_DIS
LIN {X -26.4743,Y 131.3756,Z 158,A 98.2653,B 21.4949,C -1.0012,E1 21.4868,E2 349.3836} C_DIS
LIN {X -22.832,Y 132.0595,Z 158,A 96.7328,B 21.4947,C -1.0046,E1 21.491,E2 350.9087} C_DIS
LIN {X -18.5087,Y 132.733,Z 158,A 94.8741,B 21.4947,C -1.0063,E1 21.4962,E2 352.7645} C_DIS
LIN {X -15.6475,Y 133.1,Z 158,A 93.6026,B 21.4947,C -1.0053,E1 21.4997,E2 354.0398} C_DIS
LIN {X -12.3449,Y 133.4475,Z 158,A 92.2223,B 21.4946,C -1.0077,E1 21.5035,E2 355.4144} C_DIS
LIN {X -9.6374,Y 133.6696,Z 158,A 91.0257,B 21.4946,C -1.0067,E1 21.5069,E2 356.6144} C_DIS
LIN {X -6.2955,Y 133.8693,Z 158,A 89.4713,B 21.4949,C -1.0017,E1 21.5112,E2 358.1829} C_DIS
LIN {X -2.3316,Y 133.9964,Z 158,A 87.8869,B 21.4946,C -1.007,E1 21.5156,E2 359.753} C_DIS
LIN {X 1.1903,Y 134.0121,Z 158,A 86.3072,B 21.4948,C -1.004,E1 21.52,E2 361.3409} C_DIS
LIN {X 5.1417,Y 133.9179,Z 158,A 84.6792,B 21.4946,C -1.0068,E1 21.5246,E2 362.9607} C_DIS
LIN {X 8.9978,Y 133.7163,Z 158,A 83.0736,B 21.4946,C -1.0088,E1 21.529,E2 364.5602} C_DIS
LIN {X 11.5027,Y 133.5222,Z 158,A 82.0132,B 21.4946,C -1.0093,E1 21.532,E2 365.6185} C_DIS
LIN {X 14.541,Y 133.2254,Z 158,A 80.6315,B 21.4946,C -1.0057,E1 21.5358,E2 367.009} C_DIS
LIN {X 17.8805,Y 132.8191,Z 158,A 79.2524,B 21.4946,C -1.0079,E1 21.5396,E2 368.3807} C_DIS
LIN {X 20.8345,Y 132.3874,Z 158,A 77.9863,B 21.4946,C -1.008,E1 21.5431,E2 369.6451} C_DIS
LIN {X 23.817,Y 131.8832,Z 158,A 76.6464,B 21.4946,C -1.0054,E1 21.5468,E2 370.9904} C_DIS
LIN {X 27.1934,Y 131.2293,Z 158,A 75.2073,B 21.4946,C -1.0061,E1 21.5508,E2 372.4256} C_DIS
LIN {X 30.624,Y 130.4729,Z 158,A 73.7058,B 21.4946,C -1.0053,E1 21.5548,E2 373.9269} C_DIS
LIN {X 33.2585,Y 129.8242,Z 158,A 72.5481,B 21.4947,C -1.0047,E1 21.558,E2 375.0841} C_DIS
LIN {X 36.8763,Y 128.8454,Z 158,A 70.9438,B 21.4947,C -1.0035,E1 21.5623,E2 376.6887} C_DIS
LIN {X 39.9141,Y 127.9365,Z 158,A 69.5869,B 21.4948,C -1.0023,E1 21.5659,E2 378.0457} C_DIS
LIN {X 43.1203,Y 126.8923,Z 158,A 68.1483,B 21.4948,C -1.0012,E1 21.5697,E2 379.4841} C_DIS
LIN {X 45.8308,Y 125.9366,Z 158,A 66.9067,B 21.495,C -0.9996,E1 21.573,E2 380.7273} C_DIS
LIN {X 49.3316,Y 124.609,Z 158,A 65.3221,B 21.495,C -0.9987,E1 21.5771,E2 382.3102} C_DIS
LIN {X 52.417,Y 123.3429,Z 158,A 63.8984,B 21.495,C -0.9972,E1 21.5808,E2 383.7338} C_DIS
LIN {X 55.21,Y 122.1166,Z 158,A 62.6028,B 21.4951,C -0.9961,E1 21.5841,E2 385.0287} C_DIS
LIN {X 58.2305,Y 120.7053,Z 158,A 61.1528,B 21.4952,C -0.9933,E1 21.5878,E2 386.482} C_DIS
LIN {X 61.5541,Y 119.0467,Z 158,A 59.5896,B 21.4952,C -0.9923,E1 21.5917,E2 388.0427} C_DIS
LIN {X 63.8347,Y 117.8394,Z 158,A 58.3594,B 21.4956,C -0.985,E1 21.5947,E2 389.2887} C_DIS
LIN {X 67.3672,Y 115.8558,Z 158,A 56.7618,B 21.4954,C -0.9886,E1 21.5986,E2 390.8707} C_DIS
LIN {X 70.6619,Y 113.876,Z 158,A 55.0493,B 21.4957,C -0.983,E1 21.6027,E2 392.5922} C_DIS
LIN {X 74.245,Y 111.573,Z 158,A 53.2006,B 21.4959,C -0.9788,E1 21.607,E2 394.4452} C_DIS
LIN {X 77.9064,Y 109.0478,Z 158,A 51.3232,B 21.4959,C -0.9766,E1 21.6113,E2 396.3207} C_DIS
LIN {X 81.6237,Y 106.2942,Z 158,A 49.4229,B 21.4959,C -0.9766,E1 21.6155,E2 398.2127} C_DIS
LIN {X 84.4717,Y 104.0459,Z 158,A 47.8987,B 21.496,C -0.975,E1 21.6188,E2 399.7346} C_DIS
LIN {X 87.4274,Y 101.574,Z 158,A 46.1845,B 21.4963,C -0.9687,E1 21.6225,E2 401.458} C_DIS
LIN {X 90.7003,Y 98.6625,Z 158,A 44.3299,B 21.4964,C -0.9658,E1 21.6263,E2 403.3117} C_DIS
LIN {X 93.8672,Y 95.6545,Z 158,A 42.4619,B 21.4966,C -0.9619,E1 21.6301,E2 405.1814} C_DIS
LIN {X 97.0681,Y 92.405,Z 158,A 40.5309,B 21.4967,C -0.9585,E1 21.6338,E2 407.1116} C_DIS
LIN {X 100.0057,Y 89.2174,Z 158,A 38.7332,B 21.4968,C -0.9569,E1 21.6372,E2 408.9041} C_DIS
LIN {X 102.5806,Y 86.2443,Z 158,A 37.0113,B 21.497,C -0.9511,E1 21.6403,E2 410.6325} C_DIS
LIN {X 105.1273,Y 83.122,Z 158,A 35.2405,B 21.4973,C -0.9448,E1 21.6434,E2 412.411} C_DIS
LIN {X 107.8513,Y 79.5549,Z 158,A 33.3647,B 21.4974,C -0.9421,E1 21.6466,E2 414.2834} C_DIS
LIN {X 110.3519,Y 76.0484,Z 158,A 31.5357,B 21.4976,C -0.938,E1 21.6495,E2 416.1128} C_DIS
LIN {X 112.6137,Y 72.6577,Z 158,A 29.8194,B 21.4977,C -0.9348,E1 21.6521,E2 417.8279} C_DIS
LIN {X 114.9016,Y 68.9828,Z 158,A 28.022,B 21.4978,C -0.9324,E1 21.6548,E2 419.6209} C_DIS
LIN {X 116.9705,Y 65.4126,Z 158,A 26.2984,B 21.4979,C -0.9296,E1 21.6571,E2 421.3415} C_DIS
LIN {X 118.8906,Y 61.8512,Z 158,A 24.5974,B 21.4981,C -0.9262,E1 21.6594,E2 423.041} C_DIS
LIN {X 120.4136,Y 58.8313,Z 158,A 23.1416,B 21.4983,C -0.9217,E1 21.6612,E2 424.4998} C_DIS
LIN {X 121.7614,Y 55.987,Z 158,A 21.8031,B 21.4984,C -0.9183,E1 21.6628,E2 425.8392} C_DIS
LIN {X 123.1988,Y 52.7504,Z 158,A 20.3257,B 21.4985,C -0.9157,E1 21.6644,E2 427.3141} C_DIS
LIN {X 124.4858,Y 49.6374,Z 158,A 18.8968,B 21.4987,C -0.9121,E1 21.6659,E2 428.7435} C_DIS
LIN {X 125.6607,Y 46.5823,Z 158,A 17.4827,B 21.4989,C -0.9073,E1 21.6673,E2 430.1613} C_DIS
LIN {X 126.7854,Y 43.4285,Z 158,A 16.0894,B 21.4989,C -0.9048,E1 21.6686,E2 431.5518} C_DIS
LIN {X 127.8112,Y 40.3098,Z 158,A 14.6978,B 21.4991,C -0.9012,E1 21.6698,E2 432.944} C_DIS
LIN {X 128.7549,Y 37.1857,Z 158,A 13.3422,B 21.4991,C -0.8989,E1 21.6709,E2 434.2967} C_DIS
LIN {X 129.5767,Y 34.2102,Z 158,A 12.012,B 21.4994,C -0.8944,E1 21.6718,E2 435.6301} C_DIS
LIN {X 130.4729,Y 30.624,Z 158,A 10.44,B 21.4995,C -0.8899,E1 21.6729,E2 437.2035} C_DIS
LIN {X 131.1665,Y 27.5019,Z 158,A 9.0847,B 21.4997,C -0.8863,E1 21.6737,E2 438.5593} C_DIS
LIN {X 131.7096,Y 24.7616,Z 158,A 7.9141,B 21.4997,C -0.8837,E1 21.6743,E2 439.7288} C_DIS
LIN {X 132.2147,Y 21.9016,Z 158,A 6.6313,B 21.5,C -0.8779,E1 21.6749,E2 441.0184} C_DIS
LIN {X 132.7791,Y 18.1857,Z 158,A 4.9196,B 21.5004,C -0.8678,E1 21.6756,E2 442.7457} C_DIS
LIN {X 133.2468,Y 14.343,Z 158,A 3.403,B 21.5004,C -0.8692,E1 21.6761,E2 444.2478} C_DIS
LIN {X 133.5808,Y 10.8085,Z 158,A 1.7824,B 21.5007,C -0.8594,E1 21.6765,E2 445.8835} C_DIS
LIN {X 133.8435,Y 6.8101,Z 158,A 0.2104,B 21.5007,C -0.8608,E1 21.6767,E2 447.4408} C_DIS
LIN {X 133.9775,Y 3.271,Z 158,A -1.2783,B 21.5008,C -0.8572,E1 21.6768,E2 448.9288} C_DIS
LIN {X 134.0134,Y -1.0471,Z 158,A -3.142,B 21.5011,C -0.8504,E1 21.6768,E2 450.7977} C_DIS
LIN {X 133.9441,Y -4.4716,Z 158,A -4.5474,B 21.5011,C -0.8486,E1 21.6768,E2 452.1983} C_DIS
LIN {X 133.7515,Y -8.4273,Z 158,A -6.2644,B 21.5014,C -0.842,E1 21.6765,E2 453.921} C_DIS
LIN {X 133.5021,Y -11.7404,Z 158,A -7.6103,B 21.5014,C -0.8411,E1 21.6762,E2 455.2601} C_DIS
LIN {X 133.2234,Y -14.5599,Z 158,A -8.8439,B 21.5016,C -0.8361,E1 21.6758,E2 456.4984} C_DIS
LIN {X 132.8486,Y -17.6552,Z 158,A -10.1987,B 21.5018,C -0.8308,E1 21.6754,E2 457.8582} C_DIS
LIN {X 132.3184,Y -21.2802,Z 158,A -11.7293,B 21.5019,C -0.8275,E1 21.6747,E2 459.3871} C_DIS
LIN {X 131.8857,Y -23.8033,Z 158,A -12.8515,B 21.5021,C -0.8227,E1 21.6742,E2 460.5145} C_DIS
LIN {X 131.2293,Y -27.1934,Z 158,A -14.2801,B 21.5021,C -0.8203,E1 21.6734,E2 461.9398} C_DIS
LIN {X 130.5805,Y -30.1529,Z 158,A -15.5619,B 21.5023,C -0.8169,E1 21.6726,E2 463.2221} C_DIS
LIN {X 129.7909,Y -33.3899,Z 158,A -16.9794,B 21.5025,C -0.8127,E1 21.6716,E2 464.6412} C_DIS
LIN {X 128.8454,Y -36.8763,Z 158,A -18.5226,B 21.5026,C -0.8079,E1 21.6705,E2 466.1869} C_DIS
LIN {X 127.9099,Y -40.0009,Z 158,A -19.9085,B 21.5028,C -0.804,E1 21.6694,E2 467.5742} C_DIS
LIN {X 127.0559,Y -42.6289,Z 158,A -21.0958,B 21.5029,C -0.8,E1 21.6683,E2 468.7642} C_DIS
LIN {X 125.903,Y -45.9239,Z 158,A -22.5713,B 21.503,C -0.7963,E1 21.6669,E2 470.2401} C_DIS
LIN {X 124.609,Y -49.3316,Z 158,A -24.1146,B 21.5032,C -0.7922,E1 21.6654,E2 471.7843} C_DIS
LIN {X 123.3429,Y -52.417,Z 158,A -25.5316,B 21.5033,C -0.7883,E1 21.6638,E2 473.2026} C_DIS
LIN {X 122.1794,Y -55.0694,Z 158,A -26.7673,B 21.5034,C -0.7847,E1 21.6624,E2 474.44} C_DIS
LIN {X 120.7053,Y -58.2305,Z 158,A -28.2372,B 21.5036,C -0.7813,E1 21.6607,E2 475.9099} C_DIS
LIN {X 119.0467,Y -61.5541,Z 158,A -29.8223,B 21.5037,C -0.7768,E1 21.6587,E2 477.4973} C_DIS
LIN {X 116.7031,Y -65.8883,Z 158,A -31.9797,B 21.504,C -0.7682,E1 21.6558,E2 479.6646} C_DIS
LIN {X 114.5469,Y -69.5695,Z 158,A -33.7286,B 21.504,C -0.7666,E1 21.6533,E2 481.4072} C_DIS
LIN {X 112.7317,Y -72.4739,Z 158,A -35.2483,B 21.5043,C -0.7599,E1 21.651,E2 482.9362} C_DIS
LIN {X 110.3519,Y -76.0484,Z 158,A -37.0085,B 21.5043,C -0.7584,E1 21.6482,E2 484.6901} C_DIS
LIN {X 108.361,Y -78.8593,Z 158,A -38.5368,B 21.5046,C -0.7517,E1 21.6457,E2 486.2277} C_DIS
LIN {X 105.7659,Y -82.3072,Z 158,A -40.306,B 21.5046,C -0.7505,E1 21.6428,E2 487.9905} C_DIS
LIN {X 103.4405,Y -85.2116,Z 158,A -42.0053,B 21.5049,C -0.7411,E1 21.6397,E2 489.7058} C_DIS
LIN {X 100.6942,Y -88.4404,Z 158,A -43.6887,B 21.5049,C -0.7426,E1 21.6367,E2 491.3761} C_DIS
LIN {X 98.3727,Y -91.0155,Z 158,A -45.2065,B 21.505,C -0.7372,E1 21.6338,E2 492.9005} C_DIS
LIN {X 95.4971,Y -94.0276,Z 158,A -46.9972,B 21.5052,C -0.7324,E1 21.6303,E2 494.6952} C_DIS
LIN {X 92.405,Y -97.0681,Z 158,A -48.7962,B 21.5052,C -0.7306,E1 21.6267,E2 496.4902} C_DIS
LIN {X 89.7352,Y -99.542,Z 158,A -50.4361,B 21.5055,C -0.723,E1 21.6233,E2 498.1429} C_DIS
LIN {X 86.4715,Y -102.3899,Z 158,A -52.275,B 21.5056,C -0.7195,E1 21.6194,E2 499.9828} C_DIS
LIN {X 83.122,Y -105.1273,Z 158,A -54.0476,B 21.5056,C -0.7192,E1 21.6156,E2 501.7485} C_DIS
LIN {X 79.8295,Y -107.6483,Z 158,A -55.7873,B 21.5056,C -0.717,E1 21.6117,E2 503.4865} C_DIS
LIN {X 76.8951,Y -109.7641,Z 158,A -57.361,B 21.5058,C -0.7126,E1 21.6081,E2 505.0657} C_DIS
LIN {X 73.3363,Y -112.1731,Z 158,A -59.1328,B 21.5058,C -0.7121,E1 21.604,E2 506.8318} C_DIS
LIN {X 70.4435,Y -114.012,Z 158,A -60.5905,B 21.5059,C -0.7098,E1 21.6006,E2 508.2905} C_DIS
LIN {X 67.5133,Y -115.7712,Z 158,A -62.1315,B 21.5061,C -0.7034,E1 21.5968,E2 509.8432} C_DIS
LIN {X 63.8031,Y -117.8566,Z 158,A -63.9912,B 21.5063,C -0.6984,E1 21.5923,E2 511.7102} C_DIS
LIN {X 60.3446,Y -119.6624,Z 158,A -65.5148,B 21.5062,C -0.7024,E1 21.5885,E2 513.2178} C_DIS
LIN {X 57.011,Y -121.2879,Z 158,A -67.0932,B 21.5062,C -0.7002,E1 21.5845,E2 514.7972} C_DIS
LIN {X 54.3993,Y -122.4792,Z 158,A -68.3302,B 21.5062,C -0.698,E1 21.5814,E2 516.0367} C_DIS
LIN {X 51.1813,Y -123.859,Z 158,A -69.8046,B 21.5063,C -0.6969,E1 21.5776,E2 517.51} C_DIS
LIN {X 48.0897,Y -125.0918,Z 158,A -71.2213,B 21.5063,C -0.6952,E1 21.5739,E2 518.9274} C_DIS
LIN {X 45.0891,Y -126.204,Z 158,A -72.5939,B 21.5064,C -0.6933,E1 21.5703,E2 520.302} C_DIS
LIN {X 41.87,Y -127.3086,Z 158,A -74.0325,B 21.5064,C -0.6923,E1 21.5665,E2 521.74} C_DIS
LIN {X 38.7482,Y -128.2933,Z 158,A -75.4263,B 21.5065,C -0.6909,E1 21.5628,E2 523.1345} C_DIS
LIN {X 35.6226,Y -129.1961,Z 158,A -76.8319,B 21.5065,C -0.6888,E1 21.559,E2 524.5432} C_DIS
LIN {X 31.1291,Y -130.3512,Z 158,A -78.8074,B 21.5066,C -0.6872,E1 21.5536,E2 526.5194} C_DIS
Enddeposition()
END
